(* Chamber *)
IF Config.ChamberConfigs.PhotoLumChamberConfig.IsEnabled THEN
	Chamber.FB_init(FALSE, FALSE, Config := Config.ChamberConfigs.PhotoLumChamberConfig);	
END_IF

// Chuck
IF Config.ChuckConfigs.PhotoLumChuckConfig.IsEnabled THEN
	Chuck.FB_init(FALSE, FALSE, Config := Config.ChuckConfigs.PhotoLumChuckConfig);	
END_IF 

// Axis
IF Config.AxesConfigs.Ps10OwisAxisConfig.IsEnabled THEN
	Ps10Axis.FB_init(FALSE, FALSE, Config := Config.AxesConfigs.Ps10OwisAxisConfig);	
END_IF

(* LightConfigs *) 
IF Config.LightConfigs.EvosensLightConfig.IsEnabled THEN
	EvosensLight.FB_init(FALSE, FALSE, Config := Config.LightConfigs.EvosensLightConfig);
ELSIF Config.LightConfigs.ArduinoLightConfig.IsEnabled THEN
	ArduinoLight.FB_init(FALSE, FALSE, Config := Config.LightConfigs.ArduinoLightConfig);	
END_IF

(* DistanceSensorConfigs *) 
IF Config.DistanceSensorConfigs.MicroEpsilonDistanceSensorConfig.IsEnabled THEN
	MicroEpsilonDistanceSensor.FB_init(FALSE, FALSE, Config := Config.DistanceSensorConfigs.MicroEpsilonDistanceSensorConfig);	
END_IF

IF Config.IsEnabled THEN
	_logger.Information('PhotoLum devices initialization ended...');
END_IF
END_METHOD

END_FUNCTION_BLOCK

// ---- PMShared/Hardware/Devices/Chambers/PhotoLum/PhotoLumChamber.TcPOU
{attribute 'OPC.UA.DA' := '1'}
FUNCTION_BLOCK PhotoLumChamber EXTENDS ChamberBase
VAR_INPUT
	IoChamberPhotoLum : IoChamberPhotoLum;
END_VAR
VAR_OUTPUT
END_VAR
VAR
	{attribute 'OPC.UA.DA' := '0'}
	_config : PhotoLumChamberConfig;	
	
	{attribute 'OPC.UA.DA' := '0'}
	_initDevice : BOOL;
	
	{attribute 'OPC.UA.DA' := '0'}
	_itemInit : INT;
	{attribute 'OPC.UA.DA' := '0'}
	_itemScheduler : INT;
	{attribute 'OPC.UA.DA' := '0'}
	_itemExecScheduler : INT;		
	{attribute 'OPC.UA.DA' := '0'}
	_itemRaisedProperties : INT;			
	{attribute 'OPC.UA.DA' := '0'}
	_pulseGenerator : TON;	
	
	{region 'Commands'}	
		 	
	{attribute 'OPC.UA.DA' := '0'}
	_enableCamera : BOOL;
	{attribute 'OPC.UA.DA' := '0'}
	_moveSlitDoorPositionCmd	 : BOOL;	
	{attribute 'OPC.UA.DA' := '0'}			  		   
	_raisePropertiesCmd : BOOL;	 
			
	{endregion}
	
	{attribute 'OPC.UA.DA' := '0'}
	_deliverMessages : INT;
	
	InterlockPanelsMsg : STRING(255);
	SlitDoorPositionMsg : STRING(255);
	SlitDoorOpenPositionMsg : STRING(255);
	SlitDoorClosePositionMsg : STRING(255);
	
	{attribute 'OPC.UA.DA' := '0'}
	message : STRING(255);
	
	{attribute 'OPC.UA.DA' := '0'}
	_pos : INT;	
	
	{attribute 'OPC.UA.DA' := '0'}
	tmpConcat1 : STRING;
	{attribute 'OPC.UA.DA' := '0'}
	tmpConcat2 : STRING;
	{attribute 'OPC.UA.DA' := '0'}
	tmpConcatName : STRING; 
	{attribute 'OPC.UA.DA' := '0'}
	tmpConcatDescription : STRING;
	{attribute 'OPC.UA.DA' := '0'}
	tmpConcatInterlockID : STRING;
	
	{attribute 'OPC.UA.DA' := '0'}
	_itemInterlock : UINT;
	{attribute 'OPC.UA.DA' := '0'}
	_interlockCount : UINT;			
END_VAR

SUPER^();

// Init device
InitDevice(); 

// Deliver messages
CASE _deliverMessages OF	
	EFeedbackMsgPhotoLumChamber.InterlockPanelsMsg :
		InterlockPanelsMsg := message;	
	EFeedbackMsgPhotoLumChamber.SlitDoorPositionMsg :
		SlitDoorPositionMsg := TO_STRING(SlitDoorPosition);		
	EFeedbackMsgPhotoLumChamber.SlitDoorOpenPositionMsg :
		SlitDoorOpenPositionMsg := TO_STRING(SlitDoorOpenPosition);	
	EFeedbackMsgPhotoLumChamber.SlitDoorClosePositionMsg :
		SlitDoorClosePositionMsg := TO_STRING(SlitDoorClosePosition);		
END_CASE

// Commands
MoveSlitDoorPosition(_moveSlitDoorPositionCmd, _pos); 
RaisePropertiesChanged(_raisePropertiesCmd);

IF NOT _moveSlitDoorPositionCmd AND NOT _raisePropertiesCmd THEN	
	MessageScheduler();
END_IF

METHOD FB_init : BOOL
VAR_INPUT
	bInitRetains : BOOL; // if TRUE, the retain variables are initialized (warm start / cold start)
	bInCopyCode : BOOL;  // if TRUE, the instance afterwards gets moved into the copy code (online change)
	Config : PhotoLumChamberConfig;
END_VAR
IF Config.IsEnabled THEN
	_config := Config;	

	SUPER^._chamberConfig.Name := Config.Name;
	SUPER^._chamberConfig.DeviceID := Config.DeviceID;
	SUPER^._chamberConfig.IsEnabled := Config.IsEnabled;
	SUPER^._chamberConfig.LogLevel := Config.LogLevel;
	
	SUPER^.Name := Config.Name;
	SUPER^.DeviceID := Config.DeviceID;
	
	THIS^.Family := DeviceFamily.Chamber;

	THIS^.SetReady();
	_Logger.Information(_message.Reset().Append('Init ').
							Append('{').Append(TO_STRING(THIS^.Family)).Append('} - ').
							Append('{').Append(TO_STRING(THIS^.Name)).Append('} - ').
							Append('Status : ').Append(TO_STRING(THIS^.Status)).
							ToString());										 
END_IF
END_METHOD

METHOD InitDevice
VAR_INPUT
END_VAR
IF NOT _initDevice THEN			
	_logger.Information(_message.Reset().
								Append(_config.Name).
								Append(' - init device').ToString());		
							
	_initDevice := TRUE;
	
END_IF
END_METHOD

METHOD MessageScheduler
VAR_INPUT
END_VAR
IF _pulseGenerator.Q THEN
	_pulseGenerator(IN := FALSE, PT := T#10MS);
		
	CASE _itemScheduler OF	
		0: SlitDoorPositionMsg := ' ';
		   _itemScheduler := 1;
		   
		1: ReadInterlock();
		   _itemScheduler := 2;
	
		2:  ReadSlitDoorPosition();
			_itemScheduler := 3;

		3:  ReadSlitDoorOpenPosition();
			_itemScheduler := 4;

		4:  ReadSlitDoorClosePosition();
			_itemScheduler := 0;					
	END_CASE
ELSE
	_pulseGenerator(IN := TRUE, PT := T#50MS);		
END_IF
END_METHOD

{attribute 'TcRpcEnable' := '1'}
METHOD MoveSlitDoorPosition
VAR_INPUT
	Execute : BOOL;
	Position : INT;
END_VAR
IF Execute THEN
	_logger.Information(_message.Reset().Append(_config.Name).Append(' - Move slit door position : ').Append(TO_STRING(Position)).ToString());
	
	_moveSlitDoorPositionCmd := FALSE;
		
	IF Position = ESlitDoorPosition.Open THEN
		IoChamberPhotoLum.OutputOpenSlitDoor := TRUE;
		IoChamberPhotoLum.OutputCloseSlitDoor := FALSE;
	ELSIF Position = ESlitDoorPosition.Close THEN
		IoChamberPhotoLum.OutputOpenSlitDoor := FALSE;
		IoChamberPhotoLum.OutputCloseSlitDoor := TRUE;
		
		//IsInLoadingPosition := FALSE;
	ELSE
		_logger.Error(_message.Reset().Append(_config.Name).Append(' - unknown position : ').Append(TO_STRING(Position)).ToString());
		
		//IsInLoadingPosition := FALSE;
	END_IF
				
	_itemScheduler := 0;
END_IF
END_METHOD

{attribute 'TcRpcEnable' := '1'}
METHOD RaisePropertiesChanged
VAR_INPUT
	Execute : BOOL;
END_VAR
IF Execute THEN		
	_raisePropertiesCmd := TRUE;	
		
	IF _pulseGenerator.Q THEN
		_pulseGenerator(IN := FALSE, PT := T#10MS);
		
		CASE _itemRaisedProperties OF		
			0: 	SUPER^._raisePropertiesBase := TRUE;		   
				_itemRaisedProperties := 10;
				
			10: _logger.Information(_message.Reset().Append(_config.Name).Append(' - RaisePropertiesChanged').ToString());
				_raisePropertiesCmd := FALSE;
				_itemRaisedProperties := 0;
		END_CASE	
	ELSE
		_pulseGenerator(IN := TRUE, PT := T#50MS);	
	END_IF		
END_IF
END_METHOD

METHOD ReadInterlock 
VAR_INPUT
END_VAR
VAR
	statePanel : STRING;
END_VAR
_deliverMessages := EFeedbackMsgPsdChamber.InterlockPanelsMsg;

IF _interlockCount < Const.PHOTOLUM_NUMBER_INTERLOCK_PANELS - 1 THEN
	_interlockCount := _interlockCount + 1;
ELSE
	_interlockCount := 0;
END_IF

tmpConcatName := CONCAT(_config.Interlock[_interlockCount].Name, ';');
tmpConcatDescription := CONCAT(_config.Interlock[_interlockCount].Description, ';');
tmpConcatInterlockID := CONCAT(UINT_TO_STRING(_config.Interlock[_interlockCount].InterlockID), ';');

tmpConcat1 := CONCAT(tmpConcatName, tmpConcatDescription);
tmpConcat2 := CONCAT(tmpConcat1, tmpConcatInterlockID);

IF _config.Interlock[_interlockCount].State THEN
	statePanel := 'Closed';
ELSE
	statePanel := 'Opened';
END_IF

message := CONCAT(tmpConcat2, statePanel);
END_METHOD

METHOD ReadSlitDoorClosePosition
VAR_INPUT
END_VAR
VAR
	open : BOOL;
	close : BOOL;
END_VAR
_deliverMessages := EFeedbackMsgPhotoLumChamber.SlitDoorClosePositionMsg;
SlitDoorClosePosition := IoChamberPhotoLum.InputCloseSlitDoor;
END_METHOD

METHOD ReadSlitDoorOpenPosition
VAR_INPUT
END_VAR
_deliverMessages := EFeedbackMsgPhotoLumChamber.SlitDoorOpenPositionMsg;
SlitDoorOpenPosition := IoChamberPhotoLum.InputOpenSlitDoor;
END_METHOD

METHOD ReadSlitDoorPosition
VAR_INPUT
END_VAR
VAR
	open : BOOL;
	close : BOOL;
END_VAR
_deliverMessages := EFeedbackMsgPhotoLumChamber.SlitDoorPositionMsg;

open := IoChamberPhotoLum.InputOpenSlitDoor;
close := IoChamberPhotoLum.InputCloseSlitDoor;

IF open AND NOT close THEN
	IoChamberPhotoLum.EfemInterlockSlitDoor := TRUE;	
	IoChamberPhotoLum.EfemInterlockArmExtendedEnable := TRUE;	
	SlitDoorPosition := ESlitDoorPosition.Open;	
ELSIF close AND NOT open THEN
	IoChamberPhotoLum.EfemInterlockSlitDoor := FALSE;
	IoChamberPhotoLum.EfemInterlockArmExtendedEnable := FALSE;
	SlitDoorPosition := ESlitDoorPosition.Close;
ELSIF close AND open THEN
	IoChamberPhotoLum.EfemInterlockSlitDoor := FALSE;
	IoChamberPhotoLum.EfemInterlockArmExtendedEnable := FALSE;
	SlitDoorPosition := ESlitDoorPosition.Error;	
ELSE
	IoChamberPhotoLum.EfemInterlockSlitDoor := FALSE;
	IoChamberPhotoLum.EfemInterlockArmExtendedEnable := FALSE;
	SlitDoorPosition := ESlitDoorPosition.Unknown;		
END_IF
END_METHOD

END_FUNCTION_BLOCK

// ---- PMShared/Hardware/Devices/Chucks/PhotoLum/PhotoLumChuck.TcPOU
FUNCTION_BLOCK PhotoLumChuck EXTENDS ChuckBase
VAR_INPUT
	IoChuck : IoChuckPhotoLum;
END_VAR
VAR_OUTPUT
END_VAR
VAR
	{attribute 'OPC.UA.DA' := '0'}
	_config : PhotoLumChuckConfig;
	
	{attribute 'OPC.UA.DA' := '0'}
	_deliverMessages : INT;
	
	WaferPresenceMsg : STRING(255);
	
	{attribute 'OPC.UA.DA' := '0'}
	_initDevice : BOOL;
	
	{attribute 'OPC.UA.DA' := '0'}
	_itemInit : INT;
	
	{attribute 'OPC.UA.DA' := '0'}
	_itemScheduler : INT;
	{attribute 'OPC.UA.DA' := '0'}
	_itemRaisedProperties : INT;
	{attribute 'OPC.UA.DA' := '0'}
	_pulseGenerator : TON;
	
	{region 'Commands'}
		
	{attribute 'OPC.UA.DA' := '0'}			  		   
	_clampWaferCmd : BOOL;
	{attribute 'OPC.UA.DA' := '0'}			  		   
	_releaseWaferCmd : BOOL;
	{attribute 'OPC.UA.DA' := '0'}			  		   
	_raisePropertiesCmd : BOOL;
			
	{endregion}	
		
	{attribute 'OPC.UA.DA' := '0'}	
	_size : LREAL;	
		 
	{attribute 'OPC.UA.DA' := '0'}
	message : STRING;
	{attribute 'OPC.UA.DA' := '0'}
	_waferPresenceSensorCounter : UINT;			
	
	
	
END_VAR

SUPER^();

// Init device
InitDevice(); 

// Deliver messages
CASE _deliverMessages OF		
	EFeedbackMsgPhotoLumChuck.WaferPresenceMsg :
		WaferPresenceMsg := message;		
END_CASE
	
_deliverMessages := 0;

// Commands	
ClampWafer(_clampWaferCmd, _size);
ReleaseWafer(_releaseWaferCmd, _size);
RaisePropertiesChanged(_raisePropertiesCmd);

IF (NOT _raisePropertiesCmd) THEN
	MessageScheduler();
END_IF

{attribute 'TcRpcEnable' := '1'}
METHOD ClampWafer
VAR_INPUT
	Execute : BOOL;
	Value : LREAL;
END_VAR
VAR 
	size : EWaferSize := EWaferSize.Unknown;
END_VAR
IF Execute THEN
	_logger.Information(_message.Reset().Append(_config.Name).Append(' - Clamp wafer: ').Append(TO_STRING(Value)).ToString());

	CASE LREAL_TO_INT(Value) OF
		EWaferSize._100mm : 
			IoChuck.OutputVaccum100mm := TRUE;
			IoChuck.OutputVaccum150mm := FALSE; 
			IoChuck.OutputVaccum200mm := FALSE;			
			size := EWaferSize._100mm;
			
		EWaferSize._150mm :
			IoChuck.OutputVaccum100mm := FALSE;
			IoChuck.OutputVaccum150mm := TRUE; 
			IoChuck.OutputVaccum200mm := FALSE;
			size := EWaferSize._150mm;
			
		EWaferSize._200mm :
			IoChuck.OutputVaccum100mm := FALSE;
			IoChuck.OutputVaccum150mm := FALSE; 
			IoChuck.OutputVaccum200mm := TRUE;
			size := EWaferSize._200mm;
			
		EWaferSize.Unknown:		
			size := EWaferSize.Unknown;
			_logger.Warning(_message.Reset().Append(_config.Name).Append(' - Unknown size ').ToString());
	ELSE 
		_logger.Warning(_message.Reset().Append(_config.Name).Append(' - This size: ').Append(TO_STRING(Value)).Append(' does not exist').ToString());
	END_CASE
	
	WaferSize := size;
	
	_clampWaferCmd := FALSE;
END_IF
END_METHOD

METHOD FB_init : BOOL
VAR_INPUT
	bInitRetains : BOOL; // if TRUE, the retain variables are initialized (warm start / cold start)
	bInCopyCode : BOOL;  // if TRUE, the instance afterwards gets moved into the copy code (online change)
	Config : PhotoLumChuckConfig;
END_VAR
IF Config.IsEnabled THEN
	_config := Config;
	
	SUPER^._chuckConfig.Name := Config.Name;
	SUPER^._chuckConfig.DeviceID := Config.DeviceID;
	SUPER^._chuckConfig.IsEnabled := Config.IsEnabled;
	SUPER^._chuckConfig.LogLevel := Config.LogLevel;
	
	SUPER^.Name := Config.Name;
	SUPER^.DeviceID := Config.DeviceID;
	
	THIS^.Family := DeviceFamily.Chuck;

	THIS^.SetReady();
	_Logger.Information(_message.Reset().Append('Init ').
							Append('{').Append(TO_STRING(THIS^.Family)).Append('} - ').
							Append('{').Append(TO_STRING(THIS^.Name)).Append('} - ').
							Append('Status : ').Append(TO_STRING(THIS^.Status)).
							ToString());										 
END_IF
END_METHOD

METHOD InitDevice
VAR_INPUT
END_VAR
IF NOT _initDevice THEN			
	_logger.Information(_message.Reset().
								Append(_config.Name).
								Append(' - init device').ToString());		
								
	_initDevice := TRUE;
END_IF
END_METHOD

METHOD MessageScheduler
VAR_INPUT
END_VAR
IF _pulseGenerator.Q THEN
	_pulseGenerator(IN := FALSE, PT := T#10MS);
		
	CASE _itemScheduler OF	
		0:	WaferPresenceMsg := ' ';
			_itemScheduler := 1;
	
		1:	ReadWaferPresence();
			_itemScheduler := 0;		
									
	END_CASE
ELSE
	_pulseGenerator(IN := TRUE, PT := T#100MS);	
END_IF
END_METHOD

{attribute 'TcRpcEnable' := '1'}
METHOD RaisePropertiesChanged
VAR_INPUT
	Execute : BOOL;
END_VAR
IF Execute THEN		
	_raisePropertiesCmd := TRUE;	
	
	IF _pulseGenerator.Q THEN
		_pulseGenerator(IN := FALSE, PT := T#10MS);
		
		CASE _itemRaisedProperties OF		
			0: _itemRaisedProperties := 10;
				
			10: _logger.Information(_message.Reset().Append(_config.Name).Append(' - RaisePropertiesChanged').ToString());
				_raisePropertiesCmd := FALSE;
				_itemRaisedProperties := 0;		
		END_CASE	
	ELSE
		_pulseGenerator(IN := TRUE, PT := T#100MS);	
	END_IF		
END_IF
END_METHOD

METHOD ReadWaferPresence
VAR_INPUT
END_VAR
VAR	
	waferPresence : STRING;
	diameter : STRING;
END_VAR
_deliverMessages := EFeedbackMsgPsdChuck.WaferPresenceMsg;

IF _waferPresenceSensorCounter < Const.PHOTOLUM_NUMBER_WAFER_PRESENCE_SENSORS - 1 THEN
	_waferPresenceSensorCounter := _waferPresenceSensorCounter + 1;
ELSE
	_waferPresenceSensorCounter := 0;
END_IF

diameter := TO_STRING(_config.WaferPresenceSensor[_waferPresenceSensorCounter].Diameter);

IF _config.WaferPresenceSensor[_waferPresenceSensorCounter].InputWaferPresence AND 
   _config.WaferPresenceSensor[_waferPresenceSensorCounter].Diameter = TO_UINT(_waferSize) THEN
	waferPresence := INT_TO_STRING(EMaterialPresence.Present);
ELSE
	waferPresence := INT_TO_STRING(EMaterialPresence.NotPresent);		
END_IF

message := CONCAT(CONCAT(diameter, ';'), waferPresence);
END_METHOD

{attribute 'TcRpcEnable' := '1'}
METHOD ReleaseWafer
VAR_INPUT
	Execute : BOOL;
	Value : LREAL;
END_VAR
IF Execute THEN
	_logger.Information(_message.Reset().Append(_config.Name).Append(' - release wafer: ').Append(TO_STRING(Value)).ToString());

	IF Value = EWaferSize._100mm THEN
		IoChuck.OutputVaccum100mm := FALSE;
	ELSIF Value = EWaferSize._150mm THEN		
		IoChuck.OutputVaccum150mm := FALSE; 		
	ELSIF Value = EWaferSize._200mm THEN
		IoChuck.OutputVaccum200mm := FALSE;
	ELSIF Value = EWaferSize.Unknown THEN
		_logger.Warning(_message.Reset().Append(_config.Name).Append(' - Unknown size ').ToString());
	ELSE 
		_logger.Warning(_message.Reset().Append(_config.Name).Append(' - This size: ').Append(TO_STRING(Value)).Append(' does not exist').ToString());
	END_IF

	WaferSize := EWaferSize.Unknown;
	
	_releaseWaferCmd := FALSE;
END_IF
END_METHOD

END_FUNCTION_BLOCK

// ---- PMShared/Hardware/Devices/Axes/Owis/Ps10Axis.TcPOU
FUNCTION_BLOCK Ps10Axis EXTENDS AxesBase
VAR_INPUT
END_VAR
VAR_OUTPUT
END_VAR
VAR
	{attribute 'OPC.UA.DA' := '0'}
	_config : Ps10OwisAxisConfig;
	{attribute 'OPC.UA.DA' := '0'}
	_coeAccess : CoeAccess;
	{attribute 'OPC.UA.DA' := '0'}
	_initConfigSerialCom : BOOL;	
	{attribute 'OPC.UA.DA' := '0'}
	_serialCom  : SerialCom(Prefix :='', Suffix := Const.CARRIAGE_RETURN);
	{attribute 'OPC.UA.DA' := '0'}
	_refSerialCom : REFERENCE TO SerialCom(Prefix :='', Suffix := Const.CARRIAGE_RETURN) := _serialCom;	 
	{attribute 'OPC.UA.DA' := '0'}
	_isReceived : BOOL;
	
	{attribute 'OPC.UA.DA' := '0'}
	_deliverMessages : INT;
	
	StatusMsg : STRING(255);
	AxisStatusMsg : STRING(255);
	DrivingCurrentMsg : STRING(255);
	HoldingCurrentMsg : STRING(255);
	LimitSwitchtMsg : STRING(255);
	ErrMsg : STRING(255);
	PositionMsg : STRING(255);
	CustomMsg : STRING(255);
	IsInMovingMsg : STRING(255);
	
	{region 'Commands'}	

	{attribute 'OPC.UA.DA' := '0'}
	_cmdConfigDeviceParameters : BOOL;
	{attribute 'OPC.UA.DA' := '0'}
	_cmdClearErr : BOOL;
	{attribute 'OPC.UA.DA' := '0'}
	_cmdMotorInit : BOOL;
	{attribute 'OPC.UA.DA' := '0'}
	_cmdDrivingCurrent : BOOL;
	{attribute 'OPC.UA.DA' := '0'}
	_cmdHoldingCurrent : BOOL;
	{attribute 'OPC.UA.DA' := '0'}	 
	_cmdLimitSwitch : BOOL;
	{attribute 'OPC.UA.DA' := '0'}
	_cmdReset : BOOL;
	{attribute 'OPC.UA.DA' := '0'}
	_cmdStopMotion : BOOL;		 
	{attribute 'OPC.UA.DA' := '0'}
	_cmdHomePosition : BOOL;
	{attribute 'OPC.UA.DA' := '0'}
	_cmdMoveAbsPosition : BOOL;
	{attribute 'OPC.UA.DA' := '0'}
	_customCmd : BOOL;
	{attribute 'OPC.UA.DA' := '0'}			  		   
	_cmdRaiseProperties : BOOL;	 
			
	{endregion}
		 
	{attribute 'OPC.UA.DA' := '0'}
	_initDevice : BOOL;	
		
	{attribute 'OPC.UA.DA' := '0'}
	_posToDegree : LREAL;
	{attribute 'OPC.UA.DA' := '0'}
	_cmd : STRING;
	{attribute 'OPC.UA.DA' := '0'}
	_itemScheduler : INT;
	{attribute 'OPC.UA.DA' := '0'}
	_itemRaisedProperties : INT;
	{attribute 'OPC.UA.DA' := '0'}
	_itemMove : INT;	
	{attribute 'OPC.UA.DA' := '0'}
	_itemInit : INT;
	{attribute 'OPC.UA.DA' := '0'}
	_itemdConfigDeviceParameters : INT;
	{attribute 'OPC.UA.DA' := '0'}
	_pulseGenerator : TON;
	{attribute 'OPC.UA.DA' := '0'}
	_pulseMoveGenerator : TON;	
	{attribute 'OPC.UA.DA' := '0'}
	_initPulseGenerator : TON;	
	{attribute 'OPC.UA.DA' := '0'}	
	_execPulseGenerator : TON;
	{attribute 'OPC.UA.DA' := '0'}	
	_configDeviceParamsPulseGenerator : TON;	
	
	{attribute 'OPC.UA.DA' := '0'}
	message : STRING;
	{attribute 'OPC.UA.DA' := '0'}
	lastMessage : STRING;	
	{attribute 'OPC.UA.DA' := '0'}
	stringLength : INT;
	{attribute 'OPC.UA.DA' := '0'}
	_convertDegreeToCount : LREAL := 83;
	{attribute 'OPC.UA.DA' := '0'}
	_currentAxisMode : STRING;
	{attribute 'OPC.UA.DA' := '0'}
	_currentPos : LREAL;	
	{attribute 'OPC.UA.DA' := '0'} 
	_currentPositionCounter : UINT;
	{attribute 'OPC.UA.DA' := '0'} 
	_isInMoving : BOOL;
END_VAR

IF NOT InitConfigSerialCom THEN
	ConfigureSerialCom();
ELSIF THIS^.Status = TExecutionState.Ready THEN				
	IF _refSerialCom.ErrorReceiveId = COMERROR_NOERROR THEN
		_refSerialCom(TxBuffer:= HardwareGlobalVariables.TxBufferFilterWheel, 
		 	      	  RxBuffer:= HardwareGlobalVariables.RxBufferFilterWheel);
	END_IF			

	// Init device	
	InitDevice();
		 				  	
	// Deliver messages
	IF _refSerialCom.IsReceived THEN		
		lastMessage := _refSerialCom.LastReceivedString;			
		stringLength := LEN(lastMessage);
		
		IF stringLength > 1 THEN
			message := LEFT(lastMessage, stringLength - 1);
		ELSE
			message := ' ';
		END_IF; 
				
		CASE _deliverMessages OF	
			EFeedbackMsgOwisPs10.AxisStateMsg :
				_currentAxisMode := MID(message, 1, STRING_TO_INT(AxesConst.AXIS_FILTER_WHEEL));
				AxisStatusMsg := ParseAxisStatus(_currentAxisMode);
			EFeedbackMsgOwisPs10.DrivingCurrentMsg :
				 DrivingCurrentMsg := message;
			EFeedbackMsgOwisPs10.HoldingCurrentMsg :
				 HoldingCurrentMsg := message;
			EFeedbackMsgOwisPs10.LimitSwitchMsg :
				 LimitSwitchtMsg := message;
			EFeedbackMsgOwisPs10.ErrMsg :
				 ErrMsg := message;
			EFeedbackMsgOwisPs10.PositionMsg :					
				_currentPos := STRING_TO_LREAL(message) / _convertDegreeToCount;
				PositionMsg := LREAL_TO_STRING(_currentPos);				
			EFeedbackMsgOwisPs10.CurrentPositionCounterMsg :
				_currentPositionCounter := STRING_TO_UINT(message);			
			EFeedbackMsgOwisPs10.CustomMsg :
				CustomMsg := message;						
			END_CASE
	END_IF		
			
	IF (_initDevice AND NOT _cmdClearErr AND NOT _cmdMotorInit AND NOT _cmdConfigDeviceParameters AND NOT _cmdDrivingCurrent AND NOT 
		_cmdHoldingCurrent AND NOT _cmdLimitSwitch AND NOT _cmdStopMotion AND NOT _cmdHomePosition AND NOT _cmdMoveAbsPosition AND NOT 
		_customCmd AND NOT _cmdRaiseProperties) THEN
			MessageScheduler();
	END_IF
	
	ConfigDeviceParameters(_cmdConfigDeviceParameters);
	ClearError(_cmdClearErr);
	MotorInit(_cmdMotorInit);
	SetDrivingCurrent(_cmdDrivingCurrent);
	SetHoldingCurrent(_cmdHoldingCurrent);
	SetLimitSwitch(_cmdLimitSwitch);
	Reset(_cmdReset);
	StopMotion(_cmdStopMotion);
	HomePosition(_cmdHomePosition);	
	MoveAbsPosition(_cmdMoveAbsPosition, _posToDegree);
	CustomCommand(_customCmd, _cmd);	
	RaisePropertiesChanged(_cmdRaiseProperties);	
	
END_IF

{attribute 'TcRpcEnable' := '1'}
METHOD ClearError
VAR_INPUT
	Execute : BOOL;
END_VAR
VAR
	cmd : STRING := 'ERRCLEAR';
END_VAR
IF Execute THEN
	_logger.Information(_message.Reset().Append(_config.Name).Append(' - Clear error').ToString());
	_serialCom.Send(cmd);	

	_cmdClearErr := FALSE;
END_IF
END_METHOD

METHOD ConfigDeviceParameters
VAR_INPUT
	Execute : BOOL;
END_VAR
VAR	
END_VAR
IF Execute THEN

	_cmdConfigDeviceParameters := TRUE;	

	IF _configDeviceParamsPulseGenerator.Q THEN
		_configDeviceParamsPulseGenerator(IN := FALSE, PT := T#10MS);
		
		CASE _itemdConfigDeviceParameters OF
			0:  _logger.Information(_message.Reset().Append(_config.Name).Append(' - Configure device parameters').ToString());
				_itemdConfigDeviceParameters := 1;				
								
			1: _cmdDrivingCurrent := TRUE;
				_itemdConfigDeviceParameters := 2;

			2: _cmdHoldingCurrent := TRUE;
				_itemdConfigDeviceParameters := 3;				
			
			3: _cmdLimitSwitch := TRUE;
				_itemdConfigDeviceParameters := 4;	
			
			4: _cmdMotorInit := TRUE;
				_itemdConfigDeviceParameters := 5;					
				
			5: _logger.Information(_message.Reset(). Append(_config.Name). Append(' - Configure device parameters done').ToString());	
			   _itemdConfigDeviceParameters := 0;			
			   _cmdConfigDeviceParameters := FALSE;
		END_CASE
	ELSE
		_configDeviceParamsPulseGenerator(IN := TRUE, PT := T#200MS);		
	END_IF		
END_IF
END_METHOD

METHOD ConfigureSerialCom
VAR_INPUT
END_VAR
IF _coeAccess.CoeOperation.Ready THEN
	_logger.Information(_message.Reset().Append('Start configuration com serial').ToString());
END_IF;	

_coeAccess.CoeOperation.Start();
_coeAccess(SerialCommunication := _config.SerialCommunication);
	
IF _coeAccess.CoeOperation.Done THEN
	_coeAccess.SetDone();	
 
	_Logger.Information(_message.Reset().
							Append('{').Append(TO_STRING(THIS^.Family)).Append('} : ').
							Append(' - Status : ').Append(TO_STRING(_coeAccess.Status)).ToString());	
	InitConfigSerialCom := TRUE;
END_IF
 
IF _coeAccess.CoeOperation.Error THEN	
	_coeAccess.SetError(0);
	
	_Logger.Error(_message.Reset().
							Append('{').Append(TO_STRING(THIS^.Family)).Append('} : ').
							Append(' - Status : ').Append(TO_STRING(_coeAccess.Status)).ToString());
	InitConfigSerialCom := TRUE;
END_IF

THIS^.Status := _coeAccess.Status;
State := _coeAccess.Status;
END_METHOD

{attribute 'TcRpcEnable' := '1'}
METHOD CustomCommand
VAR_INPUT
	Execute : BOOL;
	Cmd : STRING;
END_VAR
IF Execute THEN
	_logger.Information(_message.Reset().Append(_config.Name).Append(' - Custom : ').Append(Cmd).ToString());
	_deliverMessages := EFeedbackMsgOwisPs10.CustomMsg;									
	_serialCom.Send(Cmd);
	
	_customCmd := FALSE;
END_IF
END_METHOD

{attribute 'TcRpcEnable' := '1'}
METHOD ErrorMessages
VAR_INPUT
END_VAR
VAR
	cmd : STRING := '?MSG';
END_VAR
_deliverMessages := EFeedbackMsgOwisPs10.ErrMsg;	
_serialCom.Send(cmd);
END_METHOD

METHOD FB_init : BOOL
VAR_INPUT
	bInitRetains : BOOL; // if TRUE, the retain variables are initialized (warm start / cold start)
	bInCopyCode : BOOL;  // if TRUE, the instance afterwards gets moved into the copy code (online change)
	Config : Ps10OwisAxisConfig;
END_VAR
IF Config.IsEnabled THEN
	_config := Config;
	
	SUPER^._axisConfig.Name := Config.Name;
	SUPER^._axisConfig.DeviceID := Config.DeviceID;
	SUPER^._axisConfig.IsEnabled := Config.IsEnabled;
	SUPER^._axisConfig.LogLevel := Config.LogLevel;
	
	SUPER^.Name := Config.Name;
	SUPER^.DeviceID := Config.DeviceID;	
	THIS^.Family := DeviceFamily.Axes;
	
	_Logger.Information(_message.Reset().Append('Init ').
							Append('{').Append(TO_STRING(THIS^.Family)).Append('} - ').
							Append('{').Append(TO_STRING(Config.Name)).Append('}').ToString());																													
END_IF
END_METHOD

(** Axis state inquiry **)
METHOD GetAxisStatus : STRING
VAR_INPUT
END_VAR
VAR
	cmd : STRING := '?ASTAT';
END_VAR
_deliverMessages := EFeedbackMsgOwisPs10.AxisStateMsg;	
_serialCom.Send(cmd);
END_METHOD

(** Read out driving current with stepper motors in percent **)
METHOD PROTECTED GetDrivingCurrent
VAR_INPUT
END_VAR
VAR
	cmd : STRING := '?DRICUR';
END_VAR
_deliverMessages := EFeedbackMsgOwisPs10.DrivingCurrentMsg;	
_serialCom.Send(Concat(cmd, AxesConst.AXIS_FILTER_WHEEL));
END_METHOD

(** Read out holding current with stepper motor axis in percent **)
METHOD PROTECTED GetHoldingCurrent
VAR_INPUT
END_VAR
VAR
	cmd : STRING := '?HOLCUR';
END_VAR
_deliverMessages := EFeedbackMsgOwisPs10.HoldingCurrentMsg;	
_serialCom.Send(Concat(cmd, AxesConst.AXIS_FILTER_WHEEL));
END_METHOD

(** Read out limit switch mask for the axis **)
METHOD PROTECTED GetLimitSwitch
VAR_INPUT
END_VAR
VAR
	cmd : STRING := '?SMK';
END_VAR
_deliverMessages := EFeedbackMsgOwisPs10.LimitSwitchMsg;	
_serialCom.Send(Concat(cmd, AxesConst.AXIS_FILTER_WHEEL));
END_METHOD

(** Position Query **)
METHOD PROTECTED GetPosition
VAR_INPUT
END_VAR
VAR
	cmd : STRING := '?PSET';
END_VAR
_deliverMessages := EFeedbackMsgOwisPs10.PositionMsg;	
_serialCom.Send(Concat(cmd, AxesConst.AXIS_FILTER_WHEEL));
END_METHOD

{attribute 'TcRpcEnable' := '1'}
METHOD HomePosition
VAR_INPUT
	Execute : BOOL;
END_VAR
VAR
	cmd : STRING := 'REF';
END_VAR
IF Execute THEN	
	_logger.Information(_message.Reset().Append(_config.Name).Append(' - Home position : ').ToString());
	cmd := Concat(CONCAT(cmd, AxesConst.AXIS_FILTER_WHEEL), '=');	
	_serialCom.Send(Concat(cmd, '4'));
	
	_cmdHomePosition := FALSE;
END_IF
END_METHOD

PROPERTY InitConfigSerialCom : BOOL
GET
InitConfigSerialCom := _initConfigSerialCom;
END_GET
SET
_initConfigSerialCom := InitConfigSerialCom;
END_SET
END_PROPERTY

METHOD InitDevice
VAR_INPUT
END_VAR
VAR
	displayingPositionCmd : STRING := 'PWMSMODE';
	absoluteModeCmd : STRING := 'ABSOL';
	
	displayingPositionInDegree : STRING;
END_VAR
IF NOT _initDevice THEN	
	IF _initPulseGenerator.Q THEN
		_initPulseGenerator(IN := FALSE, PT := T#10MS);
		
		CASE _itemInit OF
			0:  _logger.Information(_message.Reset().Append(_config.Name).Append(' - InitDevice').ToString());
				_itemInit := 1;				
				
			1:  _cmdClearErr := TRUE;
				_itemInit := 2;
			
			2: // Absolute mode
				_serialCom.Send(CONCAT(absoluteModeCmd, AxesConst.AXIS_FILTER_WHEEL));	
				_itemInit := 10;
				
			10: _cmdConfigDeviceParameters := TRUE;	
			   _itemInit := 11;
			
			11: IF NOT _cmdConfigDeviceParameters THEN
					_itemInit := 20;
				END_IF
			
			20: GetAxisStatus();
				_itemInit := 21;
				
			21: // Displaying position in °
				displayingPositionInDegree := Concat(CONCAT(displayingPositionCmd, AxesConst.AXIS_FILTER_WHEEL), '=');
				_serialCom.Send(CONCAT(displayingPositionInDegree, '3'));				
				_itemInit := 22;													
				
			22:  IF _currentAxisMode = 'R' THEN	
					_itemInit := 30;	
				ELSE			
					_logger.Error(_message.Reset().Append(_config.Name).Append(' - Axis status : ').
								  Append(_currentAxisMode).ToString());
					_itemInit := 40;				  
			    END_IF							
				
			30:  GetPosition();
				_itemInit := 31;	
				
			31: _posToDegree := _currentPos;
				_itemInit := 40;
				
			40: _logger.Information(_message.Reset(). Append(_config.Name). Append(' - InitDevice done').ToString());	
				_itemInit := 0;			
				_initDevice	:= TRUE;
		END_CASE
	ELSE
		_initPulseGenerator(IN := TRUE, PT := T#100MS);		
	END_IF		
END_IF
END_METHOD

PROPERTY IsInMoving : bool
GET
IsInMoving := _isInMoving;
END_GET
SET
_isInMoving := IsInMoving;
END_SET
END_PROPERTY

METHOD MessageScheduler
VAR_INPUT
END_VAR
IF _pulseGenerator.Q THEN
	_pulseGenerator(IN := FALSE, PT := T#10MS);
	
	CASE _itemScheduler OF				
		0:	GetAxisStatus();
			_itemScheduler := 1;
						
		1:	GetPosition();
			_itemScheduler := 0;			
	END_CASE		
ELSE
	_pulseGenerator(IN := TRUE, PT := T#100MS);		
END_IF
END_METHOD

{attribute 'TcRpcEnable' := '1'}
METHOD MotorInit
VAR_INPUT
	Execute : BOOL;
END_VAR
VAR	
	cmd : STRING := 'INIT';
END_VAR
IF Execute THEN
	_logger.Information(_message.Reset().Append(_config.Name).Append(' - Enable the motor power stage').ToString());
	_serialCom.Send(Concat(cmd, AxesConst.AXIS_FILTER_WHEEL));	

	_cmdMotorInit := FALSE;	
END_IF
END_METHOD

{attribute 'TcRpcEnable' := '1'}
METHOD PROTECTED MoveAbsPosition 
VAR_INPUT
	Execute : BOOL;
	Position : LREAL;
END_VAR
VAR
	cmdSet : STRING := 'PSET';
	cmdGo : STRING := 'PGO';
	cmdCnt : STRING := '?CNT';
	cmd : STRING;	
END_VAR
IF Execute THEN

	_cmdMoveAbsPosition := TRUE;
	_posToDegree := Position;	
	
	IF _pulseMoveGenerator.Q THEN
		_pulseMoveGenerator(IN := FALSE, PT := T#10MS);
	
		CASE _itemMove OF
			0:	_logger.Information(_message.Reset().Append(_config.Name).Append(' - Move absolute position : ').
													 Append(TO_STRING(_posToDegree)).Append(' °').ToString());
								
				cmd := Concat(CONCAT(cmdSet, AxesConst.AXIS_FILTER_WHEEL), '=');				
				_serialCom.Send(CONCAT(cmd, LREAL_TO_STRING(_posToDegree * _convertDegreeToCount)));				
				_itemMove := 1;						
				
			1:  _serialCom.Send(Concat(cmdGo, AxesConst.AXIS_FILTER_WHEEL));											
				_itemMove := 2;	
				
			2:  _deliverMessages := EFeedbackMsgOwisPs10.CurrentPositionCounterMsg;	
				IF _currentPositionCounter <> (_posToDegree * _convertDegreeToCount) THEN					
					_serialCom.Send(Concat(cmdCnt, AxesConst.AXIS_FILTER_WHEEL));
					IsInMovingMsg := BOOL_TO_STRING(TRUE);	
				ELSE
					IsInMovingMsg := BOOL_TO_STRING(FALSE);	
					_itemMove := 3;	
				END_IF
								
			3: _cmdMoveAbsPosition := FALSE;
				_itemMove := 0;
			
		END_CASE			
	ELSE
		_pulseMoveGenerator(IN := TRUE, PT := T#100MS);	
	END_IF

END_IF
END_METHOD

METHOD PRIVATE ParseAxisStatus : STRING
VAR_INPUT
	CurrentAxisMode : STRING;
END_VAR
VAR
	Description : STRING;
END_VAR
IF CurrentAxisMode = 'I' THEN
	Description := 'Axis is not initialized';
ELSIF CurrentAxisMode = 'O' THEN
	Description := 'Axis is disabled';
ELSIF CurrentAxisMode = 'R' THEN
	Description := 'Axis initialized and ready';
ELSIF CurrentAxisMode = 'T' THEN
	Description := 'Axis is positioning in trapezoidal profile';
ELSIF CurrentAxisMode = 'V' THEN
	Description := 'Axis is operating in velocity mode';
ELSIF CurrentAxisMode = 'P' THEN
	Description := 'Reference motion is in progress';
ELSIF CurrentAxisMode = 'F' THEN
	Description := 'Axis is releasing a limit switch';
ELSIF CurrentAxisMode = 'L' THEN
	Description := 'Axis has been disabled after approaching a hardware limit switch(MINSTOP, MAXSTOP)';
ELSIF CurrentAxisMode = 'B' THEN
	Description := 'Aaxis has been stopped after approaching a brake switch(MINDEC, MAXDEC)';
ELSIF CurrentAxisMode = 'A' THEN
	Description := 'Axis has been disabled after limit switch error';
ELSIF CurrentAxisMode = 'M' THEN
	Description := 'Axis has been disabled after motion-controller error';
ELSIF CurrentAxisMode = 'Z' THEN
	Description := 'Axis has been disabled after timeout error';
ELSIF CurrentAxisMode = 'H' THEN
	Description := 'Phase initialization active (step motor axis)';
ELSIF CurrentAxisMode = 'U' THEN
	Description := 'Axis not enabled';
ELSIF CurrentAxisMode = 'E' THEN
	Description := 'Axis has been disabled after motion error';
ELSIF CurrentAxisMode = '?' THEN
	Description := 'Error, unknown state of axis';
ELSE
	Description := 'Unknown error';
END_IF

ParseAxisStatus := Description;
END_METHOD

{attribute 'TcRpcEnable' := '1'}
METHOD RaisePropertiesChanged
VAR_INPUT
	Execute : BOOL;
END_VAR
IF Execute THEN
	IF THIS^.Status <> TExecutionState.Ready THEN	
		_cmdRaiseProperties := FALSE;
		RETURN;
	END_IF	

	_cmdRaiseProperties := TRUE;
	
	IF _pulseGenerator.Q THEN
		_pulseGenerator(IN := FALSE, PT := T#10MS);	

		CASE _itemRaisedProperties OF
			0:  StateMsg := ' ';
				AxisStatusMsg := ' ';
				ErrMsg := ' ';
				PositionMsg := ' ';
				CustomMsg := ' ';
				
				_itemRaisedProperties := 10;
			
			10:  GetPosition();
				_itemRaisedProperties := 11;
			
			11:  GetAxisStatus();
				 _itemRaisedProperties := 12;
				 
			12:  ErrorMessages();
				 _itemRaisedProperties := 20;			
				 
			20:  _logger.Information(_message.Reset().Append(_config.Name).Append(' - PS10 Axis RaisePropertiesChanged').ToString());
				_cmdRaiseProperties := FALSE;				
				_itemRaisedProperties := 0;
			
		END_CASE
	ELSE
		_pulseGenerator(IN := TRUE, PT := T#100MS);	
	END_IF
END_IF
END_METHOD

{attribute 'TcRpcEnable' := '1'}
METHOD Reset
VAR_INPUT
	Execute : BOOL;
END_VAR
VAR
	cmd : STRING := 'RESETMB';
END_VAR
IF Execute THEN
	_logger.Information(_message.Reset().Append(_config.Name).Append(' - Release reset main board').ToString());
	_serialCom.Send(cmd);	
	
	_cmdReset := FALSE;
END_IF
END_METHOD

{attribute 'TcRpcEnable' := '1'}
METHOD SetDrivingCurrent
VAR_INPUT
	Execute : BOOL;
END_VAR
VAR
	cmdSet : STRING := 'DRICUR';
	cmd : STRING;
END_VAR
IF Execute THEN
	_logger.Information(_message.Reset().Append(_config.Name).Append(' - driving current with stepper motor: ').
		Append(TO_STRING(AxesConst.FW_DRIVING_CURRENT_IN_PERCENT)).ToString());
	
	cmd := Concat(CONCAT(cmdSet, AxesConst.AXIS_FILTER_WHEEL), '=');
	_serialCom.Send(CONCAT(cmd, TO_STRING(AxesConst.FW_DRIVING_CURRENT_IN_PERCENT)));	

	_cmdDrivingCurrent := FALSE;	
END_IF
END_METHOD

{attribute 'TcRpcEnable' := '1'}
METHOD SetHoldingCurrent
VAR_INPUT
	Execute : BOOL;
END_VAR
VAR
	cmdSet : STRING := 'HOLCUR';
	cmd : STRING;
END_VAR
IF Execute THEN
	_logger.Information(_message.Reset().Append(_config.Name).Append(' - holding current with stepper motor axes: ').
		Append(TO_STRING(AxesConst.FW_HOLDING_CURRENT_IN_PERCENT)).ToString());
	
	cmd := Concat(CONCAT(cmdSet, AxesConst.AXIS_FILTER_WHEEL), '=');
	_serialCom.Send(CONCAT(cmd, TO_STRING(AxesConst.FW_HOLDING_CURRENT_IN_PERCENT)));	

	_cmdHoldingCurrent := FALSE;	
END_IF
END_METHOD

{attribute 'TcRpcEnable' := '1'}
METHOD SetLimitSwitch
VAR_INPUT
	Execute : BOOL;
END_VAR
VAR
	cmdSet : STRING := 'SMK';
	cmd : STRING;
END_VAR
IF Execute THEN
	_logger.Information(_message.Reset().Append(_config.Name).Append(' -  limit switch mask for the axis: ').
		Append(TO_STRING(AxesConst.FW_LIMIT_SWITCH_MASK)).ToString());
	
	cmd := Concat(CONCAT(cmdSet, AxesConst.AXIS_FILTER_WHEEL), '=');
	_serialCom.Send(CONCAT(cmd, TO_STRING(AxesConst.FW_LIMIT_SWITCH_MASK)));	

	_cmdLimitSwitch := FALSE;	
END_IF
END_METHOD

{attribute 'TcRpcEnable' := '1'}
METHOD StopMotion
VAR_INPUT
	Execute : BOOL;
END_VAR
VAR
	cmd : STRING := 'STOP1';
END_VAR
IF Execute THEN	
	_logger.Information(_message.Reset().Append(_config.Name).Append(' - Stop motion').ToString());
	_serialCom.Send(cmd);
	
	_cmdStopMotion := FALSE;
END_IF
END_METHOD

END_FUNCTION_BLOCK

// ---- PMShared/Hardware/Devices/Lights/Evosens/EvosensLight.TcPOU
{attribute 'OPC.UA.DA' := '1'}
FUNCTION_BLOCK EvosensLight EXTENDS LightBase
VAR_INPUT
END_VAR
VAR_OUTPUT
END_VAR
VAR
	{attribute 'OPC.UA.DA' := '0'}
	_config : EvosensLightConfig;	
	{attribute 'OPC.UA.DA' := '0'}
	_coeAccess : CoeAccess;	
	{attribute 'OPC.UA.DA' := '0'}
	_initConfigSerialCom : BOOL;	
	{attribute 'OPC.UA.DA' := '0'}
	_suffix : STRING := Const.CR_LF;
	{attribute 'OPC.UA.DA' := '0'}
	_serialCom  : SerialCom(Prefix :='', Suffix := _suffix);
	{attribute 'OPC.UA.DA' := '0'}
	_refSerialCom : REFERENCE TO SerialCom(Prefix :='', Suffix := _suffix) := _serialCom;		 
	{attribute 'OPC.UA.DA' := '0'}
	_isReceived : BOOL;
	
	{attribute 'OPC.UA.DA' := '0'}
	_deliverMessages : INT;
		
	StatusMsg : STRING(255);
	SwitchOnMsg : STRING(255);
	PowerMsg : STRING(255);
	IntensityMsg : STRING(255);	
	TemperatureMsg : STRING(255);
	LightSourcesMsg : STRING(255);
	TimeLightSourceMsg  : STRING(255);
	CustomMsg : STRING(255);
		
	{region 'Commands'}
	
	{attribute 'OPC.UA.DA' := '0'}
	_setSwitchOnCmd : BOOL;
	{attribute 'OPC.UA.DA' := '0'}
	_getSwitchOnCmd : BOOL;
	{attribute 'OPC.UA.DA' := '0'}
	_setPowerCmd : BOOL;
	{attribute 'OPC.UA.DA' := '0'}
	_getPowerCmd : BOOL;
	{attribute 'OPC.UA.DA' := '0'}
	_setIntensityCmd : BOOL;
	{attribute 'OPC.UA.DA' := '0'}
	_getIntensityCmd : BOOL;
	{attribute 'OPC.UA.DA' := '0'}
	_getTimeLightSourceCmd : BOOL;
	{attribute 'OPC.UA.DA' := '0'}
	_getLightSourcesCmd : BOOL;
	{attribute 'OPC.UA.DA' := '0'}
	_customCmd : BOOL;
	{attribute 'OPC.UA.DA' := '0'}			  		   
	_raisePropertiesCmd : BOOL;
	
	{attribute 'OPC.UA.DA' := '0'}
	_lightId : UINT; 
	{attribute 'OPC.UA.DA' := '0'}
	_switchOn : BOOL;
	{attribute 'OPC.UA.DA' := '0'}
	_setPower : LREAL;
	{attribute 'OPC.UA.DA' := '0'}
	_setIntensity : LREAL;
	{attribute 'OPC.UA.DA' := '0'}
	_cmd : STRING;	
		 
	{endregion}			
	
	{attribute 'OPC.UA.DA' := '0'}
	_initDevice : BOOL;	
	 
	{attribute 'OPC.UA.DA' := '0'}
	_lightSources : ARRAY [0..Const.PHOTOLUM_NUMBER_LIGHT_SOURCE] OF STRING(255);  
	
	{attribute 'OPC.UA.DA' := '0'}
	_itemScheduler : INT;
	{attribute 'OPC.UA.DA' := '0'}
	_itemInitScheduler : INT;
	{attribute 'OPC.UA.DA' := '0'}
	_itemExecScheduler : INT;		
	{attribute 'OPC.UA.DA' := '0'}
	_itemRaisedProperties : INT;			
	{attribute 'OPC.UA.DA' := '0'}
	_pulseGenerator : TON;	
	{attribute 'OPC.UA.DA' := '0'}
	_initPulseGenerator : TON;	
	{attribute 'OPC.UA.DA' := '0'}	
	_execPulseGenerator : TON;	
	
	{attribute 'OPC.UA.DA' := '0'}
	message : STRING;
	{attribute 'OPC.UA.DA' := '0'}
	lastMessage : STRING;	
	{attribute 'OPC.UA.DA' := '0'}
	sSubStr4 : STRING(4) := '';			
	{attribute 'OPC.UA.DA' := '0'}
	stringLength : INT;
	{attribute 'OPC.UA.DA' := '0'}
	_numberOfElements : DINT;
	{attribute 'OPC.UA.DA' := '0'}
	_indexNumberOfElements : INT;
END_VAR

IF NOT InitConfigSerialCom THEN
	ConfigureSerialCom();
ELSIF THIS^.Status = TExecutionState.Ready THEN
	SUPER^();	

	IF _refSerialCom.ErrorReceiveId = COMERROR_NOERROR THEN
		_refSerialCom(TxBuffer:= HardwareGlobalVariables.TxBufferLight, 
		 	      	  RxBuffer:= HardwareGlobalVariables.RxBufferLight);
	END_IF				  
	
	// Init device
	InitDevice(); 				  				 	
	
	IF StateMsg <> ANY_TO_STRING(State) THEN
		StateMsg := ANY_TO_STRING(State);
	END_IF
	
	// Deliver messages
	IF _refSerialCom.IsReceived THEN	
		lastMessage := _refSerialCom.LastReceivedString;			
		stringLength := LEN(lastMessage);
		
		IF stringLength > 2 THEN
			message := LEFT(lastMessage, stringLength - 2);
		ELSE
			message := ' ';
		END_IF; 	
			
		CASE _deliverMessages OF			
			EFeedbackMsgArduinoLight.SwitchOnMsg :
				SwitchOnMsg := message;	
			EFeedbackMsgArduinoLight.PowerMsg :
				PowerMsg := message;	
			EFeedbackMsgArduinoLight.IntensityMsg :
				IntensityMsg := message;	
			EFeedbackMsgArduinoLight.TemperatureMsg :
				TemperatureMsg := message;	
			EFeedbackMsgArduinoLight.LightSourcesMsg :
				LightSourcesMsg := message;			
				_logger.Information(_message.Reset().Append('LightSourcesMsg: ').Append(LightSourcesMsg).ToString());	
			EFeedbackMsgArduinoLight.TimeLightSourceMsg :
				TimeLightSourceMsg := message;	
			EFeedbackMsgArduinoLight.CustomMsg :
				CustomMsg := message;	
		END_CASE
	
		_deliverMessages := 0;
	END_IF								   							   	
		
	SetSwitchOn(_setSwitchOnCmd, TO_STRING(_lightId), _switchOn); 
	GetSwitchOn(_getSwitchOnCmd, TO_STRING(_lightId));
	SetPower(_setPowerCmd, TO_STRING(_lightId), _setPower);
	GetPower(_getPowerCmd, TO_STRING(_lightId));
	//SetIntensity(_setIntensityCmd, TO_STRING(_lightId), _setIntensity);
	//GetIntensity(_getIntensityCmd, TO_STRING(_lightId));
	GetTimeLightSource(_getTimeLightSourceCmd, TO_STRING(_lightId));
	GetLightSources(_getLightSourcesCmd);
	CustomCommand(_customCmd, _cmd);
	RaisePropertiesChanged(_raisePropertiesCmd, TO_STRING(_lightId));
	
	IF _initDevice AND NOT _setSwitchOnCmd AND NOT _getSwitchOnCmd AND NOT _setPowerCmd AND NOT _getPowerCmd AND NOT _setIntensityCmd AND NOT _getIntensityCmd
	   AND NOT _getTimeLightSourceCmd AND NOT _getLightSourcesCmd AND NOT _customCmd AND NOT _raisePropertiesCmd THEN
		MessageScheduler();
	END_IF
END_IF

METHOD ConfigureSerialCom
VAR_INPUT
END_VAR
IF _coeAccess.CoeOperation.Ready THEN
	_logger.Information(_message.Reset().Append('Start configuration com serial').ToString());
END_IF;	

_coeAccess.CoeOperation.Start();
_coeAccess(SerialCommunication := _config.SerialCommunication);
	
IF _coeAccess.CoeOperation.Done THEN
	_coeAccess.SetDone();	
	
	_Logger.Information(_message.Reset().
							Append('{').Append(TO_STRING(THIS^.Family)).Append('} : ').
							Append(' - Status : ').Append(TO_STRING(_coeAccess.Status)).ToString());	
	InitConfigSerialCom := TRUE;
END_IF
 
IF _coeAccess.CoeOperation.Error THEN	
	_coeAccess.SetError(0);
	
	_Logger.Error(_message.Reset().
							Append('{').Append(TO_STRING(THIS^.Family)).Append('} : ').
							Append(' - Status : ').Append(TO_STRING(_coeAccess.Status)).ToString());
	InitConfigSerialCom := TRUE;
END_IF

THIS^.Status := _coeAccess.Status;
State := _coeAccess.Status;
END_METHOD

{attribute 'TcRpcEnable' := '1'}
(** Custom command **)
METHOD CustomCommand
VAR_INPUT
	Execute : BOOL;
	Cmd : STRING;
END_VAR
IF Execute THEN
	_logger.Information(_message.Reset().Append(_config.Name).Append(' - Custom command : ').Append(Cmd).ToString());	
	_deliverMessages := EFeedbackMsgArduinoLight.CustomMsg;														
	_serialCom.Send(Cmd);	
	_customCmd := FALSE;
END_IF
END_METHOD

METHOD FB_init : BOOL
VAR_INPUT
	bInitRetains : BOOL; // if TRUE, the retain variables are initialized (warm start / cold start)
	bInCopyCode : BOOL;  // if TRUE, the instance afterwards gets moved into the copy code (online change)
	Config : EvosensLightConfig;
END_VAR
IF Config.IsEnabled THEN
	_config := Config;
	
	SUPER^._lightConfig.Name := Config.Name;
	SUPER^._lightConfig.DeviceID := Config.DeviceID;
	SUPER^._lightConfig.IsEnabled := Config.IsEnabled;
	SUPER^._lightConfig.LogLevel := Config.LogLevel;
	
	SUPER^.Name := Config.Name;
	SUPER^.DeviceID := Config.DeviceID;	
	THIS^.Family := DeviceFamily.Light;
		
	_Logger.Information(_message.Reset().Append('Init ').
							Append('{').Append(TO_STRING(THIS^.Family)).Append('} - ').
							Append('{').Append(TO_STRING(Config.Name)).Append('}').ToString());																													
END_IF
END_METHOD

{attribute 'TcRpcEnable' := '1'}
METHOD GetIntensity
VAR_INPUT
	Execute : BOOL;
	LightId : STRING;
END_VAR
VAR
	cmd : STRING := '*amps ';
END_VAR
IF Execute THEN	
	_deliverMessages := EFeedbackMsgArduinoLight.IntensityMsg;
	_serialCom.Send(CONCAT(cmd, LightId));
	
	_getIntensityCmd := FALSE;
END_IF
END_METHOD

METHOD GetLightSources
VAR_INPUT
	Execute: BOOL;
END_VAR
VAR
	cmd : STRING := '*light';
END_VAR
IF Execute THEN
	_logger.Information(_message.Reset().Append(_config.Name).Append(' - GetLightSources').ToString());
	_deliverMessages := EFeedbackMsgArduinoLight.LightSourcesMsg;
	_serialCom.Send(cmd);	
	
	_getLightSourcesCmd := FALSE;
END_IF
END_METHOD

{attribute 'TcRpcEnable' := '1'}
METHOD GetPower
VAR_INPUT
	Execute : BOOL;
	LightId : STRING;
END_VAR
VAR
	cmd : STRING := '*power ';
END_VAR
IF Execute THEN	
	_deliverMessages := EFeedbackMsgArduinoLight.PowerMsg;
	_serialCom.Send(CONCAT(cmd, LightId));
	
	 _getPowerCmd := FALSE;
END_IF
END_METHOD

{attribute 'TcRpcEnable' := '1'}
METHOD GetSwitchOn
VAR_INPUT
	Execute : BOOL;
	LightId : STRING;
END_VAR
VAR
	cmd : STRING := '*switch ';
END_VAR
IF Execute THEN	
	_deliverMessages := EFeedbackMsgArduinoLight.SwitchOnMsg;
	_serialCom.Send(CONCAT(cmd, LightId));
				
	_getSwitchOnCmd := FALSE;	
END_IF
END_METHOD

METHOD GetTemperature
VAR_INPUT
	LightId : STRING;
END_VAR
VAR
	cmd : STRING := '*temp ';
END_VAR
_deliverMessages := EFeedbackMsgArduinoLight.TemperatureMsg;
_serialCom.Send(CONCAT(cmd, LightId));
END_METHOD

METHOD GetTimeLightSource
VAR_INPUT
	Execute: BOOL;
	LightId : STRING;
END_VAR
VAR
	cmd : STRING := '*time ';
END_VAR
IF Execute THEN
	_logger.Information(_message.Reset().Append(_config.Name).Append(' - GetTimeLightSource - ').Append(LightId).ToString());
	_deliverMessages := EFeedbackMsgArduinoLight.TimeLightSourceMsg;
	_serialCom.Send(CONCAT(cmd, LightId));	
	
	_getTimeLightSourceCmd := FALSE;
END_IF
END_METHOD

PROPERTY InitConfigSerialCom : BOOL
GET
InitConfigSerialCom := _initConfigSerialCom;
END_GET
SET
_initConfigSerialCom := InitConfigSerialCom;
END_SET
END_PROPERTY

METHOD InitDevice
VAR_INPUT
END_VAR
VAR
	numElements : INT := 0;
    commaPos : INT;
    tempStr : STRING; 
	Separator : STRING := ',';
END_VAR
IF NOT _initDevice THEN	
	IF _initPulseGenerator.Q THEN
		_initPulseGenerator(IN := FALSE, PT := T#10MS);
			
		CASE _itemInitScheduler OF					
			0:	_logger.Information(_message.Reset().Append(_config.Name).Append(' - Init device').ToString());
				//_getLightSourcesCmd := TRUE;
				_itemInitScheduler := 50;
			
			1:	IF LightSourcesMsg <> '' THEN				
					tempStr := LightSourcesMsg;
					WHILE (LEN(tempStr) > 0) DO
						commaPos := FIND(tempStr, Separator);
						IF commaPos > 0 THEN
							_lightSources[numElements] := LEFT(tempStr, commaPos - 1);						
							tempStr := RIGHT(tempStr, LEN(tempStr) - commaPos);
						ELSE
							_lightSources[numElements] := tempStr;
							tempStr := ''; 
						END_IF
						_logger.Information(_message.Reset().Append(_config.Name).Append(' - ').Append(TO_STRING(numElements)).Append(': ').Append(_lightSources[numElements]).ToString());
						numElements := numElements + 1;						
					END_WHILE
														
					IF (numElements - 1) <> 0 THEN
						_numberOfElements := numElements;
						//_itemInitScheduler := 10; GVA
						_itemInitScheduler := 50;
					ELSE
						_itemInitScheduler := 40;	
					END_IF				
					
					_deliverMessages := -1;
				END_IF
			
			10: IF (_indexNumberOfElements >= 0) AND (_indexNumberOfElements < _numberOfElements) THEN
					tempStr := CONCAT(_lightSources[_indexNumberOfElements], ' 0');
					_serialCom.Send(CONCAT('*power ', tempStr));				
					_logger.Information(_message.Reset().Append(_config.Name).Append(' - ').Append(_lightSources[_indexNumberOfElements]).Append(' - Power: 0').ToString());	
					_indexNumberOfElements := _indexNumberOfElements + 1;
					
				ELSE
					_indexNumberOfElements := 0;
					_itemInitScheduler := 11;					
				END_IF	
			
			11: IF (_indexNumberOfElements >= 0) AND (_indexNumberOfElements < _numberOfElements) THEN
					tempStr := CONCAT(_lightSources[_indexNumberOfElements], ' 1');
					_serialCom.Send(CONCAT('*swit ', tempStr));
					_logger.Information(_message.Reset().Append(_config.Name).Append(' - ').Append(_lightSources[_indexNumberOfElements]).Append(' - Switch ON').ToString());
					_indexNumberOfElements := _indexNumberOfElements + 1;					
				ELSE
					_indexNumberOfElements := 0;
					_itemInitScheduler := 50;
				END_IF	

			41: _logger.Error(_message.Reset().Append(_config.Name).Append(' - numElements is empty: ').ToString());
				_itemInitScheduler := 50;	
		
			50: _initDevice := TRUE;
				_itemInitScheduler := 0;	
				_logger.Information(_message.Reset().Append(_config.Name).Append(' - Init device done').ToString());	
		END_CASE
	ELSE
		_initPulseGenerator(IN := TRUE, PT := T#100MS);		
	END_IF	
END_IF
END_METHOD

METHOD MessageScheduler
VAR_INPUT
END_VAR
VAR
	
END_VAR
IF _pulseGenerator.Q THEN
	_pulseGenerator(IN := FALSE, PT := T#10MS);
		
	CASE _itemScheduler OF					
		0:	_getSwitchOnCmd := TRUE;
			_itemScheduler := 1;
			
		1:	_getPowerCmd := TRUE;
			_itemScheduler := 2;
			
		2:  //GetTemperature(_lightID);			
			_itemScheduler := 10;
			
		10: IF _lightId > 0 AND _lightId < Const.PHOTOLUM_NUMBER_LIGHT_SOURCE THEN
				_lightId := _lightId + 1;				
			ELSE
				_lightId := 1;
			END_IF
			
			
			_itemScheduler := 0;
									
	END_CASE
ELSE
	_pulseGenerator(IN := TRUE, PT := T#250MS);		
END_IF


IF _pulseIsAliveGenerator.Q THEN
	_pulseIsAliveGenerator(IN := FALSE, PT := T#10MS);
		
	IsAlive();	
ELSE
	_pulseIsAliveGenerator(IN := TRUE, PT := T#1000MS);		
END_IF
END_METHOD

{attribute 'TcRpcEnable' := '1'}
METHOD RaisePropertiesChanged
VAR_INPUT
	Execute : BOOL;
	LightId : STRING;
END_VAR
VAR
	numElements : INT := 0;
    commaPos : INT;
    tempStr : STRING; 
	Separator : STRING := ',';
END_VAR
IF Execute THEN
	_raisePropertiesCmd := TRUE;
	IF LightId <> '' THEN
		_lightId := STRING_TO_UINT(LightId);
	END_IF
	
	IF _pulseGenerator.Q THEN
		_pulseGenerator(IN := FALSE, PT := T#10MS);	

		CASE _itemRaisedProperties OF
			0:  SwitchOnMsg := ' ';
				PowerMsg := ' ';		
				IntensityMsg := ' ';
				LightSourcesMsg := ' ';		
				TimeLightSourceMsg := ' ';		
				_itemRaisedProperties := 1;					

			1:  IF _lightId > 0 AND _lightId <= Const.PHOTOLUM_NUMBER_LIGHT_SOURCE THEN
					_itemRaisedProperties := 50;	
				ELSE
					_itemRaisedProperties := 40;	
				END_IF  
				
			10: _getSwitchOnCmd := TRUE;													
				_itemRaisedProperties := 11;
				
			11: IF SwitchOnMsg <> ' ' THEN
					_itemRaisedProperties := 12;
				END_IF	
				
			12: _getPowerCmd := TRUE;													
				_itemRaisedProperties := 13;
				
			13: IF PowerMsg <> ' ' THEN
					_itemRaisedProperties := 16;
				END_IF
							
			16: _getTimeLightSourceCmd := TRUE;													
				_itemRaisedProperties := 17;
				
			17: IF TimeLightSourceMsg <> ' ' THEN
					_itemRaisedProperties := 50;
				END_IF
			
			40: _logger.Error(_message.Reset().Append(_config.Name).Append(' - RaisePropertiesChanged - LightId is empty').ToString());
				_itemRaisedProperties := 50;
			
			50:  _logger.Information(_message.Reset().Append(_config.Name).Append(' - RaisePropertiesChanged').ToString());
				_raisePropertiesCmd := FALSE;				
				_itemRaisedProperties := 0;
			
		END_CASE
	ELSE
		_pulseGenerator(IN := TRUE, PT := T#100MS);	
	END_IF
END_IF
END_METHOD

{attribute 'TcRpcEnable' := '1'}
METHOD SetIntensity
VAR_INPUT
	Execute : BOOL;
	LightId : STRING;
	Intensity : LREAL;
END_VAR
VAR
	cmd : STRING := '*amps ';
	tmpConcatLightIdIntensity : STRING;
END_VAR
IF Execute THEN	
	_setIntensityCmd := TRUE;
	_setIntensity := Intensity; 
	IF LightId <> '' THEN
		_lightId := STRING_TO_UINT(LightId);
	END_IF
	
	IF _execPulseGenerator.Q THEN
		_execPulseGenerator(IN := FALSE, PT := T#10MS);
			
		CASE _itemExecScheduler OF
			0:  IF _lightId > 0 AND _lightId <= Const.PHOTOLUM_NUMBER_LIGHT_SOURCE THEN
					_itemExecScheduler := 10;	
				ELSE
					_itemExecScheduler := 40;	
				END_IF
				
				_deliverMessages := -1;

			10: tmpConcatLightIdIntensity := CONCAT(CONCAT(TO_STRING(_lightId), ' '), TO_STRING(Intensity));

				_logger.Information(_message.Reset().Append(_config.Name).Append(' - ').Append(TO_STRING(_lightId)).Append(' - SetIntensity : ').Append(TO_STRING(_lightId)).Append(' - ').Append(TO_STRING(Intensity)).ToString());
				_serialCom.Send(CONCAT(cmd, TO_STRING(tmpConcatLightIdIntensity)));
				_itemExecScheduler := 11;
			
			11:  _getIntensityCmd := TRUE;
				_itemExecScheduler := 50;
			
			40: _logger.Error(_message.Reset().Append(_config.Name).Append(' - SetIntensity - light id is not valid').ToString());
				_itemExecScheduler := 50;
		
			50:  _setIntensityCmd := FALSE;	
				_itemExecScheduler := 0;		
								
		END_CASE
	ELSE
		_execPulseGenerator(IN := TRUE, PT := T#100MS);	
	END_IF
END_IF
END_METHOD

{attribute 'TcRpcEnable' := '1'}
METHOD SetPower
VAR_INPUT
	Execute : BOOL;
	LightId : STRING;
	Power : LREAL;
END_VAR
VAR
	cmd : STRING := '*power ';
	tmpConcatLightIdPower : STRING;
END_VAR
IF Execute THEN	
	_setPowerCmd := TRUE;		
	_setPower := Power;	
	IF LightId <> '' THEN
		_lightId := STRING_TO_UINT(LightId);
	END_IF
	
	IF _execPulseGenerator.Q THEN
		_execPulseGenerator(IN := FALSE, PT := T#10MS);
			
		CASE _itemExecScheduler OF
			0: IF _lightId > 0 AND _lightId <= Const.PHOTOLUM_NUMBER_LIGHT_SOURCE THEN
					_itemExecScheduler := 10;	
				ELSE
					_itemExecScheduler := 40;	
				END_IF
				
				_deliverMessages := -1;

			10: tmpConcatLightIdPower := CONCAT(CONCAT(TO_STRING(_lightId), ' '), TO_STRING(Power));

				_logger.Information(_message.Reset().Append(_config.Name).Append(' - ').Append(TO_STRING(_lightId)).Append(' - SetPower : ').Append(TO_STRING(Power)).ToString());
				_serialCom.Send(CONCAT(cmd, TO_STRING(tmpConcatLightIdPower)));
				_itemExecScheduler := 11;
			
			11:  _getPowerCmd := TRUE;
				_itemExecScheduler := 50;
			
			40: _logger.Error(_message.Reset().Append(_config.Name).Append(' - SetPower - light id is not valid').ToString());
				_itemExecScheduler := 50;
	
			50:  _setPowerCmd := FALSE;	
				_itemExecScheduler := 0;		
								
		END_CASE
	ELSE
		_execPulseGenerator(IN := TRUE, PT := T#100MS);	
	END_IF
END_IF
END_METHOD

{attribute 'TcRpcEnable' := '1'}
METHOD SetSwitchOn
VAR_INPUT
	Execute : BOOL;	
	LightId : STRING;
	SwitchOn : BOOL;
END_VAR
VAR
	cmd : STRING := '*switch ';
	tmpConcatLightIdSwitchOn : STRING;
	tmp : STRING;
	switchOnValue : STRING;
END_VAR
IF Execute THEN	
	_setSwitchOnCmd := TRUE;	
	_switchOn := SwitchOn; 
	
	IF LightId <> '' THEN
		_lightId := STRING_TO_UINT(LightId);
	END_IF	
	
	IF _execPulseGenerator.Q THEN
		_execPulseGenerator(IN := FALSE, PT := T#10MS);
			
		CASE _itemExecScheduler OF
			0:  IF _lightId > 0 AND _lightId <= Const.PHOTOLUM_NUMBER_LIGHT_SOURCE THEN
					_itemExecScheduler := 10;	
				ELSE
					_itemExecScheduler := 40;	
				END_IF
				
				_deliverMessages := -1;

			10:	IF _switchOn THEN
					switchOnValue := 'ON';
				ELSE
					switchOnValue := 'OFF';
				END_IF
				tmpConcatLightIdSwitchOn := CONCAT(CONCAT(TO_STRING(_lightId), ' '), TO_STRING(switchOnValue));
				
				_logger.Information(_message.Reset().Append(_config.Name).Append(' - ').Append(TO_STRING(_lightId)).Append(' - SwitchOn : ').Append(TO_STRING(switchOnValue)).ToString());
				tmp := CONCAT(cmd, TO_STRING(tmpConcatLightIdSwitchOn));
				_serialCom.Send(tmp);
				_itemExecScheduler := 11;
			
			11:  _getSwitchOnCmd := TRUE;
				_itemExecScheduler := 50;
				
			40: _logger.Error(_message.Reset().Append(_config.Name).Append(' - SwitchOn - light id is not valid').ToString());
				_itemExecScheduler := 50;
				
			50:  _setSwitchOnCmd := FALSE;	
				_switchOn := FALSE;
				_itemExecScheduler := 0;		
								
		END_CASE
	ELSE
		_execPulseGenerator(IN := TRUE, PT := T#200MS);	
	END_IF
END_IF
END_METHOD

END_FUNCTION_BLOCK

// ---- PMShared/Hardware/Devices/Lights/LightBase.TcPOU
FUNCTION_BLOCK ABSTRACT LightBase EXTENDS TExecution IMPLEMENTS IDevice
VAR_INPUT
END_VAR
VAR_OUTPUT
END_VAR
VAR
	{attribute 'OPC.UA.DA' := '0'}
	_name : STRING;
	{attribute 'OPC.UA.DA' := '0'}
	_deviceID : STRING;				
	{attribute 'OPC.UA.DA' := '0'}	
	_family : DeviceFamily;	
	{attribute 'OPC.UA.DA' := '0'}
	_logger : Logger;
	{attribute 'OPC.UA.DA' := '0'}
	_message : StringBuilder;
	{attribute 'OPC.UA.DA' := '0'}
	_lightConfig : DeviceConfiguration;	
	
	{attribute 'OPC.UA.DA' := '0'}
	_lifeTimeCount : UINT;
	{attribute 'OPC.UA.DA' := '0'}
	_notifyIsAlive : BOOL;
	{attribute 'OPC.UA.DA' := '0'}
	_pulseIsAliveGenerator : TON;				
		
	StateMsg : STRING(255);
	IsAliveMsg : STRING(255);
END_VAR

// Check if it's still alive	
IF _notifyIsAlive THEN
	IsAliveMsg := TO_STRING(_lifeTimeCount);
	_notifyIsAlive := FALSE;
END_IF

IF HardwareGlobalVariables.LightState <> State THEN
	HardwareGlobalVariables.LightState := State;
	StateMsg := ANY_TO_STRING(State);		
END_IF

MessageSchedulerBase();

PROPERTY DeviceID : STRING
GET
DeviceID := _deviceID;
END_GET
SET
_deviceID := DeviceID;
END_SET
END_PROPERTY

PROPERTY Family : DeviceFamily
GET
Family := _family;
END_GET
SET
_family := Family;
END_SET
END_PROPERTY

METHOD IsAlive
VAR_INPUT
END_VAR
_notifyIsAlive := TRUE;

IF _lifeTimeCount < 5 THEN
	_lifeTimeCount := _lifeTimeCount + 1;
ELSE
	_lifeTimeCount := 1;
END_IF
END_METHOD

METHOD MessageSchedulerBase
VAR_INPUT
END_VAR
IF _pulseIsAliveGenerator.Q THEN
	_pulseIsAliveGenerator(IN := FALSE, PT := T#10MS);
		
	IsAlive();	
ELSE
	_pulseIsAliveGenerator(IN := TRUE, PT := T#1000MS);		
END_IF
END_METHOD

PROPERTY Name : STRING
GET
Name := _name;
END_GET
SET
_name := Name;
END_SET
END_PROPERTY

METHOD ABSTRACT SetIntensity
VAR_INPUT
	Execute : BOOL;
	LightId : STRING;
	Intensity : LREAL;
END_VAR
END_METHOD

END_FUNCTION_BLOCK

// ---- PMShared/Hardware/Devices/Lights/Arduino/ArduinoLight.TcPOU
{attribute 'OPC.UA.DA' := '1'}
FUNCTION_BLOCK ArduinoLight EXTENDS LightBase
VAR_INPUT
END_VAR
VAR_OUTPUT
END_VAR
VAR
	{attribute 'OPC.UA.DA' := '0'}
	_config : ArduinoLightConfig;	
	{attribute 'OPC.UA.DA' := '0'}
	_coeAccess : CoeAccess;	
	{attribute 'OPC.UA.DA' := '0'}
	_initConfigSerialCom : BOOL;	
	{attribute 'OPC.UA.DA' := '0'}
	_suffix : STRING := Const.CR_LF;
	{attribute 'OPC.UA.DA' := '0'}
	_serialCom  : SerialCom(Prefix :='', Suffix := _suffix);
	{attribute 'OPC.UA.DA' := '0'}
	_refSerialCom : REFERENCE TO SerialCom(Prefix :='', Suffix := _suffix) := _serialCom;		 
	{attribute 'OPC.UA.DA' := '0'}
	_isReceived : BOOL;
	
	{attribute 'OPC.UA.DA' := '0'}
	_deliverMessages : INT;
		
	StatusMsg : STRING(255);
	SwitchOnMsg : STRING(255);
	PowerMsg : STRING(255);
	IntensityMsg : STRING(255);	
	TemperatureMsg : STRING(255);
	LightSourcesMsg : STRING(255);
	TimeLightSourceMsg  : STRING(255);
	CustomMsg : STRING(255);
		
	{region 'Commands'}
	
	{attribute 'OPC.UA.DA' := '0'}
	_setSwitchOnCmd : BOOL;
	{attribute 'OPC.UA.DA' := '0'}
	_getSwitchOnCmd : BOOL;
	{attribute 'OPC.UA.DA' := '0'}
	_setPowerCmd : BOOL;
	{attribute 'OPC.UA.DA' := '0'}
	_getPowerCmd : BOOL;
	{attribute 'OPC.UA.DA' := '0'}
	_setIntensityCmd : BOOL;
	{attribute 'OPC.UA.DA' := '0'}
	_getIntensityCmd : BOOL;
	{attribute 'OPC.UA.DA' := '0'}
	_getTimeLightSourceCmd : BOOL;
	{attribute 'OPC.UA.DA' := '0'}
	_getLightSourcesCmd : BOOL;
	{attribute 'OPC.UA.DA' := '0'}
	_customCmd : BOOL;
	{attribute 'OPC.UA.DA' := '0'}			  		   
	_raisePropertiesCmd : BOOL;
	
	{attribute 'OPC.UA.DA' := '0'}
	_lightId : STRING; 
	{attribute 'OPC.UA.DA' := '0'}
	_switchOn : BOOL;
	{attribute 'OPC.UA.DA' := '0'}
	_setPower : LREAL;
	{attribute 'OPC.UA.DA' := '0'}
	_setIntensity : LREAL;
	{attribute 'OPC.UA.DA' := '0'}
	_cmd : STRING;	
		 
	{endregion}			
	
	{attribute 'OPC.UA.DA' := '0'}
	_initDevice : BOOL;	
	 
	{attribute 'OPC.UA.DA' := '0'}
	_lightSources : ARRAY [0..Const.PHOTOLUM_NUMBER_LIGHT_SOURCE] OF STRING(255);  
	
	{attribute 'OPC.UA.DA' := '0'}
	_itemScheduler : INT;
	{attribute 'OPC.UA.DA' := '0'}
	_itemInitScheduler : INT;
	{attribute 'OPC.UA.DA' := '0'}
	_itemExecScheduler : INT;		
	{attribute 'OPC.UA.DA' := '0'}
	_itemRaisedProperties : INT;			
	{attribute 'OPC.UA.DA' := '0'}
	_pulseGenerator : TON;	
	{attribute 'OPC.UA.DA' := '0'}
	_initPulseGenerator : TON;	
	{attribute 'OPC.UA.DA' := '0'}	
	_execPulseGenerator : TON;	
	
	{attribute 'OPC.UA.DA' := '0'}
	message : STRING;
	{attribute 'OPC.UA.DA' := '0'}
	lastMessage : STRING;	
	{attribute 'OPC.UA.DA' := '0'}
	sSubStr4 : STRING(4) := '';			
	{attribute 'OPC.UA.DA' := '0'}
	stringLength : INT;
	{attribute 'OPC.UA.DA' := '0'}
	_numberOfElements : DINT;
	{attribute 'OPC.UA.DA' := '0'}
	_indexNumberOfElements : INT;
END_VAR

IF NOT InitConfigSerialCom THEN
	ConfigureSerialCom();
ELSIF THIS^.Status = TExecutionState.Ready THEN
	SUPER^();	

	IF _refSerialCom.ErrorReceiveId = COMERROR_NOERROR THEN
		_refSerialCom(TxBuffer:= HardwareGlobalVariables.TxBufferLight, 
		 	      	  RxBuffer:= HardwareGlobalVariables.RxBufferLight);
	END_IF				  
	
	// Init device
	InitDevice();		  				 
	
	IF StateMsg <> ANY_TO_STRING(State) THEN
		StateMsg := ANY_TO_STRING(State);
	END_IF
	
	// Deliver messages
	IF _refSerialCom.IsReceived THEN	
		lastMessage := _refSerialCom.LastReceivedString;			
		stringLength := LEN(lastMessage);
		
		IF stringLength > 2 THEN
			message := LEFT(lastMessage, stringLength - 2);
		ELSE
			message := ' ';
		END_IF; 	
			
		CASE _deliverMessages OF			
			EFeedbackMsgArduinoLight.SwitchOnMsg :
				SwitchOnMsg := message;	
			EFeedbackMsgArduinoLight.PowerMsg :
				PowerMsg := message;	
			EFeedbackMsgArduinoLight.IntensityMsg :
				IntensityMsg := message;	
			EFeedbackMsgArduinoLight.TemperatureMsg :
				TemperatureMsg := message;	
			EFeedbackMsgArduinoLight.LightSourcesMsg :
				LightSourcesMsg := message;			
				_logger.Information(_message.Reset().Append('LightSourcesMsg: ').Append(LightSourcesMsg).ToString());	
			EFeedbackMsgArduinoLight.TimeLightSourceMsg :
				TimeLightSourceMsg := message;	
			EFeedbackMsgArduinoLight.CustomMsg :
				CustomMsg := message;	
		END_CASE
		
		_deliverMessages := 0;
	END_IF								   							   	
		
	SetSwitchOn(_setSwitchOnCmd, _lightId, _switchOn); 
	GetSwitchOn(_getSwitchOnCmd, _lightId);
	SetPower(_setPowerCmd, _lightId, _setPower);
	GetPower(_getPowerCmd, _lightId);
	SetIntensity(_setIntensityCmd, _lightId, _setIntensity);
	GetIntensity(_getIntensityCmd, _lightId);
	GetTimeLightSource(_getTimeLightSourceCmd, _lightId);
	GetLightSources(_getLightSourcesCmd);
	CustomCommand(_customCmd, _cmd);
	RaisePropertiesChanged(_raisePropertiesCmd, _lightId);
	
	IF _initDevice AND NOT _setSwitchOnCmd AND NOT _getSwitchOnCmd AND NOT _setPowerCmd AND NOT _getPowerCmd AND NOT _setIntensityCmd AND NOT _getIntensityCmd
	   AND NOT _getTimeLightSourceCmd AND NOT _getLightSourcesCmd AND NOT _customCmd AND NOT _raisePropertiesCmd THEN
		MessageScheduler();
	END_IF
END_IF

METHOD ConfigureSerialCom
VAR_INPUT
END_VAR
IF _coeAccess.CoeOperation.Ready THEN
	_logger.Information(_message.Reset().Append('Start configuration com serial').ToString());
END_IF;	

_coeAccess.CoeOperation.Start();
_coeAccess(SerialCommunication := _config.SerialCommunication);
	
IF _coeAccess.CoeOperation.Done THEN
	_coeAccess.SetDone();	
	
	_Logger.Information(_message.Reset().
							Append('{').Append(TO_STRING(THIS^.Family)).Append('} : ').
							Append(' - Status : ').Append(TO_STRING(_coeAccess.Status)).ToString());	
	InitConfigSerialCom := TRUE;
END_IF
 
IF _coeAccess.CoeOperation.Error THEN	
	_coeAccess.SetError(0);
	
	_Logger.Error(_message.Reset().
							Append('{').Append(TO_STRING(THIS^.Family)).Append('} : ').
							Append(' - Status : ').Append(TO_STRING(_coeAccess.Status)).ToString());
	InitConfigSerialCom := TRUE;
END_IF

THIS^.Status := _coeAccess.Status;
State := _coeAccess.Status;
END_METHOD

{attribute 'TcRpcEnable' := '1'}
(** Custom command **)
METHOD CustomCommand
VAR_INPUT
	Execute : BOOL;
	Cmd : STRING;
END_VAR
IF Execute THEN
	_logger.Information(_message.Reset().Append(_config.Name).Append(' - Custom command : ').Append(Cmd).ToString());	
	_deliverMessages := EFeedbackMsgArduinoLight.CustomMsg;														
	_serialCom.Send(Cmd);	
	_customCmd := FALSE;
END_IF
END_METHOD

METHOD FB_init : BOOL
VAR_INPUT
	bInitRetains : BOOL; // if TRUE, the retain variables are initialized (warm start / cold start)
	bInCopyCode : BOOL;  // if TRUE, the instance afterwards gets moved into the copy code (online change)
	Config : ArduinoLightConfig;
END_VAR
IF Config.IsEnabled THEN
	_config := Config;
	
	SUPER^._lightConfig.Name := Config.Name;
	SUPER^._lightConfig.DeviceID := Config.DeviceID;
	SUPER^._lightConfig.IsEnabled := Config.IsEnabled;
	SUPER^._lightConfig.LogLevel := Config.LogLevel;
	
	SUPER^.Name := Config.Name;
	SUPER^.DeviceID := Config.DeviceID;	
	THIS^.Family := DeviceFamily.Light;
		
	_Logger.Information(_message.Reset().Append('Init ').
							Append('{').Append(TO_STRING(THIS^.Family)).Append('} - ').
							Append('{').Append(TO_STRING(Config.Name)).Append('}').ToString());																													
END_IF
END_METHOD

{attribute 'TcRpcEnable' := '1'}
METHOD GetIntensity
VAR_INPUT
	Execute : BOOL;
	LightId : STRING;
END_VAR
VAR
	cmd : STRING := '*amps ';
END_VAR
IF Execute THEN	
	_deliverMessages := EFeedbackMsgArduinoLight.IntensityMsg;
	_lightId := LightId;
	_serialCom.Send(CONCAT(cmd, TO_STRING(_lightId)));
	
	_getIntensityCmd := FALSE;
END_IF
END_METHOD

METHOD GetLightSources
VAR_INPUT
	Execute: BOOL;
END_VAR
VAR
	cmd : STRING := '*list';
END_VAR
IF Execute THEN
	_logger.Information(_message.Reset().Append(_config.Name).Append(' - GetLightSources').ToString());
	_deliverMessages := EFeedbackMsgArduinoLight.LightSourcesMsg;
	_serialCom.Send(cmd);	
	
	_getLightSourcesCmd := FALSE;
END_IF
END_METHOD

{attribute 'TcRpcEnable' := '1'}
METHOD GetPower
VAR_INPUT
	Execute : BOOL;
	LightId : STRING;
END_VAR
VAR
	cmd : STRING := '*power ';
END_VAR
IF Execute THEN	
	_deliverMessages := EFeedbackMsgArduinoLight.PowerMsg;
	_lightId := LightId;
	_serialCom.Send(CONCAT(cmd, TO_STRING(_lightId)));
	
	 _getPowerCmd := FALSE;
END_IF
END_METHOD

{attribute 'TcRpcEnable' := '1'}
METHOD GetSwitchOn
VAR_INPUT
	Execute : BOOL;
	LightId : STRING;
END_VAR
VAR
	cmd : STRING := '*swit ';
END_VAR
IF Execute THEN	
	_deliverMessages := EFeedbackMsgArduinoLight.SwitchOnMsg;
	_lightId := LightId;
	_serialCom.Send(CONCAT(cmd, TO_STRING(_lightId)));
				
	_getSwitchOnCmd := FALSE;	
END_IF
END_METHOD

METHOD GetTemperature
VAR_INPUT
	LightId : STRING;
END_VAR
VAR
	cmd : STRING := '*temp ';
END_VAR
_deliverMessages := EFeedbackMsgArduinoLight.TemperatureMsg;
_lightId := LightId;
_serialCom.Send(CONCAT(cmd, _lightId));
END_METHOD

METHOD GetTimeLightSource
VAR_INPUT
	Execute: BOOL;
	LightId : STRING;
END_VAR
VAR
	cmd : STRING := '*time ';
END_VAR
IF Execute THEN
	_lightId := LightId;
	_logger.Information(_message.Reset().Append(_config.Name).Append(' - GetTimeLightSource - ').Append(TO_STRING(_lightId)).ToString());
	_deliverMessages := EFeedbackMsgArduinoLight.TimeLightSourceMsg;
	_serialCom.Send(CONCAT(cmd, _lightId));	
	
	_getTimeLightSourceCmd := FALSE;
END_IF
END_METHOD

PROPERTY InitConfigSerialCom : BOOL
GET
InitConfigSerialCom := _initConfigSerialCom;
END_GET
SET
_initConfigSerialCom := InitConfigSerialCom;
END_SET
END_PROPERTY

METHOD InitDevice
VAR_INPUT
END_VAR
VAR
	numElements : INT := 0;
    commaPos : INT;
    tempStr : STRING; 
	Separator : STRING := ',';
END_VAR
IF NOT _initDevice THEN	
	IF _initPulseGenerator.Q THEN
		_initPulseGenerator(IN := FALSE, PT := T#10MS);
			
		CASE _itemInitScheduler OF					
			0:	_logger.Information(_message.Reset().Append(_config.Name).Append(' - Init device').ToString());
				//_getLightSourcesCmd := TRUE;
				_itemInitScheduler := 50;
			
			1:	IF LightSourcesMsg <> '' THEN				
					tempStr := LightSourcesMsg;
					WHILE (LEN(tempStr) > 0) DO
						commaPos := FIND(tempStr, Separator);
						IF commaPos > 0 THEN
							_lightSources[numElements] := LEFT(tempStr, commaPos - 1);						
							tempStr := RIGHT(tempStr, LEN(tempStr) - commaPos);
						ELSE
							_lightSources[numElements] := tempStr;
							tempStr := ''; 
						END_IF
						_logger.Information(_message.Reset().Append(_config.Name).Append(' - ').Append(TO_STRING(numElements)).Append(': ').Append(_lightSources[numElements]).ToString());
						numElements := numElements + 1;						
					END_WHILE
														
					IF (numElements - 1) <> 0 THEN
						_numberOfElements := numElements;
						//_itemInitScheduler := 10; GVA
						_itemInitScheduler := 50;
					ELSE
						_itemInitScheduler := 40;	
					END_IF				
					
					_deliverMessages := -1;
				END_IF
			
			10: IF (_indexNumberOfElements >= 0) AND (_indexNumberOfElements < _numberOfElements) THEN
					tempStr := CONCAT(_lightSources[_indexNumberOfElements], ' 0');
					_serialCom.Send(CONCAT('*power ', tempStr));				
					_logger.Information(_message.Reset().Append(_config.Name).Append(' - ').Append(_lightSources[_indexNumberOfElements]).Append(' - Power: 0').ToString());	
					_indexNumberOfElements := _indexNumberOfElements + 1;
					
				ELSE
					_indexNumberOfElements := 0;
					_itemInitScheduler := 11;					
				END_IF	
			
			11: IF (_indexNumberOfElements >= 0) AND (_indexNumberOfElements < _numberOfElements) THEN
					tempStr := CONCAT(_lightSources[_indexNumberOfElements], ' 1');
					_serialCom.Send(CONCAT('*swit ', tempStr));
					_logger.Information(_message.Reset().Append(_config.Name).Append(' - ').Append(_lightSources[_indexNumberOfElements]).Append(' - Switch ON').ToString());
					_indexNumberOfElements := _indexNumberOfElements + 1;					
				ELSE
					_indexNumberOfElements := 0;
					_itemInitScheduler := 50;
				END_IF	

			41: _logger.Error(_message.Reset().Append(_config.Name).Append(' - numElements is empty: ').ToString());
				_itemInitScheduler := 50;	
		
			50: _initDevice := TRUE;
				_itemInitScheduler := 0;	
				_logger.Information(_message.Reset().Append(_config.Name).Append(' - Init device done').ToString());	
		END_CASE
	ELSE
		_initPulseGenerator(IN := TRUE, PT := T#100MS);		
	END_IF	
END_IF
END_METHOD

METHOD MessageScheduler
VAR_INPUT
END_VAR
IF _pulseGenerator.Q THEN
	_pulseGenerator(IN := FALSE, PT := T#10MS);
		
	CASE _itemScheduler OF					
		0:	IF _lightID <> '' THEN
				//GetTemperature(_lightID);
			END_IF
				
			_itemScheduler := 0;		
	END_CASE
ELSE
	_pulseGenerator(IN := TRUE, PT := T#100MS);		
END_IF


IF _pulseIsAliveGenerator.Q THEN
	_pulseIsAliveGenerator(IN := FALSE, PT := T#10MS);
		
	IsAlive();	
ELSE
	_pulseIsAliveGenerator(IN := TRUE, PT := T#1000MS);		
END_IF
END_METHOD

{attribute 'TcRpcEnable' := '1'}
METHOD RaisePropertiesChanged
VAR_INPUT
	Execute : BOOL;
	LightId : STRING;
END_VAR
VAR
	numElements : INT := 0;
    commaPos : INT;
    tempStr : STRING; 
	Separator : STRING := ',';
END_VAR
IF Execute THEN
	_raisePropertiesCmd := TRUE;
	_lightId := LightId;
	
	IF _pulseGenerator.Q THEN
		_pulseGenerator(IN := FALSE, PT := T#10MS);	

		CASE _itemRaisedProperties OF
			0:  SwitchOnMsg := ' ';
				PowerMsg := ' ';		
				IntensityMsg := ' ';
				LightSourcesMsg := ' ';		
				TimeLightSourceMsg := ' ';		
				_itemRaisedProperties := 1;					

			1:  IF _lightId <> '' THEN
					_itemRaisedProperties := 10;	
				ELSE
					_itemRaisedProperties := 40;	
				END_IF
				
			10: _getSwitchOnCmd := TRUE;													
				_itemRaisedProperties := 11;
				
			11: IF SwitchOnMsg <> ' ' THEN
					_itemRaisedProperties := 12;
				END_IF	
				
			12: _getPowerCmd := TRUE;													
				_itemRaisedProperties := 13;
				
			13: IF PowerMsg <> ' ' THEN
					_itemRaisedProperties := 14;
				END_IF
				
			14: _getIntensityCmd := TRUE;													
				_itemRaisedProperties := 15;
				
			15: IF IntensityMsg <> ' ' THEN
					_itemRaisedProperties := 16;
				END_IF
			
			16: _getTimeLightSourceCmd := TRUE;													
				_itemRaisedProperties := 17;
				
			17: IF TimeLightSourceMsg <> ' ' THEN
					_itemRaisedProperties := 50;
				END_IF
			
			40: _logger.Error(_message.Reset().Append(_config.Name).Append(' - RaisePropertiesChanged - LightId is empty').ToString());
				_itemRaisedProperties := 50;
			
			50:  _logger.Information(_message.Reset().Append(_config.Name).Append(' - RaisePropertiesChanged').ToString());
				_raisePropertiesCmd := FALSE;				
				_itemRaisedProperties := 0;
			
		END_CASE
	ELSE
		_pulseGenerator(IN := TRUE, PT := T#50MS);	
	END_IF
END_IF
END_METHOD

{attribute 'TcRpcEnable' := '1'}
METHOD SetIntensity
VAR_INPUT
	Execute : BOOL;
	LightId : STRING;
	Intensity : LREAL;
END_VAR
VAR
	cmd : STRING := '*amps ';
	tmpConcatLightIdIntensity : STRING;
END_VAR
IF Execute THEN	
	_setIntensityCmd := TRUE;
	_lightId := LightId;
	_setIntensity := Intensity; 
	
	IF _execPulseGenerator.Q THEN
		_execPulseGenerator(IN := FALSE, PT := T#10MS);
			
		CASE _itemExecScheduler OF
			0:  IF _lightId <> '' THEN
					_itemExecScheduler := 10;	
				ELSE
					_itemExecScheduler := 40;	
				END_IF
				
				_deliverMessages := -1;

			10: _lightId := LightId;
				tmpConcatLightIdIntensity := CONCAT(CONCAT(_lightId, ' '), TO_STRING(Intensity));

				_logger.Information(_message.Reset().Append(_config.Name).Append(' - ').Append(_lightId).Append(' - SetIntensity : ').Append(TO_STRING(_lightId)).Append(' - ').Append(TO_STRING(Intensity)).ToString());
				_serialCom.Send(CONCAT(cmd, TO_STRING(tmpConcatLightIdIntensity)));
				_itemExecScheduler := 11;
			
			11:  _getIntensityCmd := TRUE;
				_itemExecScheduler := 50;
			
			40: _logger.Error(_message.Reset().Append(_config.Name).Append(' - SetIntensity - LightId is empty').ToString());
				_itemExecScheduler := 50;
		
			50:  _setIntensityCmd := FALSE;	
				_itemExecScheduler := 0;		
								
		END_CASE
	ELSE
		_execPulseGenerator(IN := TRUE, PT := T#100MS);	
	END_IF
END_IF
END_METHOD

{attribute 'TcRpcEnable' := '1'}
METHOD SetPower
VAR_INPUT
	Execute : BOOL;
	LightId : STRING;
	Power : LREAL;
END_VAR
VAR
	cmd : STRING := '*power ';
	tmpConcatLightIdPower : STRING;
END_VAR
IF Execute THEN	
	_setPowerCmd := TRUE;	
	_lightId := LightId;
	_setPower := Power;	
	
	IF _execPulseGenerator.Q THEN
		_execPulseGenerator(IN := FALSE, PT := T#10MS);
			
		CASE _itemExecScheduler OF
			0:  IF _lightId <> '' THEN
					_itemExecScheduler := 10;	
				ELSE
					_itemExecScheduler := 40;	
				END_IF
				
				_deliverMessages := -1;

			10: _lightId := LightId;
				tmpConcatLightIdPower := CONCAT(CONCAT(_lightId, ' '), TO_STRING(Power));

				_logger.Information(_message.Reset().Append(_config.Name).Append(' - ').Append(_lightId).Append(' - SetPower : ').Append(TO_STRING(Power)).ToString());
				_serialCom.Send(CONCAT(cmd, TO_STRING(tmpConcatLightIdPower)));
				_itemExecScheduler := 11;
			
			11:  _getPowerCmd := TRUE;
				_itemExecScheduler := 50;
			
			40: _logger.Error(_message.Reset().Append(_config.Name).Append(' - SetPower - LightId is empty').ToString());
				_itemExecScheduler := 50;
	
			50:  _setPowerCmd := FALSE;	
				_itemExecScheduler := 0;		
								
		END_CASE
	ELSE
		_execPulseGenerator(IN := TRUE, PT := T#100MS);	
	END_IF
END_IF
END_METHOD

{attribute 'TcRpcEnable' := '1'}
METHOD SetSwitchOn
VAR_INPUT
	Execute : BOOL;	
	LightId : STRING;
	SwitchOn : BOOL;
END_VAR
VAR
	cmd : STRING := '*swit ';
	tmpConcatLightIdSwitchOn : STRING;
	tmp : STRING;
	switchOnValue : STRING;
END_VAR
IF Execute THEN	
	_setSwitchOnCmd := TRUE;	
	_switchOn := SwitchOn; 
	_lightId := LightId;
	
	IF _execPulseGenerator.Q THEN
		_execPulseGenerator(IN := FALSE, PT := T#10MS);
			
		CASE _itemExecScheduler OF
			0:  IF _lightId <> '' THEN
					_itemExecScheduler := 10;	
				ELSE
					_itemExecScheduler := 40;	
				END_IF
				
				_deliverMessages := -1;

			10:	_lightId := LightId;				
			
				IF _switchOn THEN
					switchOnValue := '1';
				ELSE
					switchOnValue := '0';
				END_IF
				tmpConcatLightIdSwitchOn := CONCAT(CONCAT(_lightId, ' '), TO_STRING(switchOnValue));
				
				_logger.Information(_message.Reset().Append(_config.Name).Append(' - ').Append(_lightId).Append(' - SwitchOn : ').Append(TO_STRING(switchOnValue)).ToString());
				tmp := CONCAT(cmd, TO_STRING(tmpConcatLightIdSwitchOn));
				_serialCom.Send(tmp);
				_itemExecScheduler := 11;
			
			11:  _getSwitchOnCmd := TRUE;
				_itemExecScheduler := 50;
				
			40: _logger.Error(_message.Reset().Append(_config.Name).Append(' - SwitchOn - LightId is empty').ToString());
				_itemExecScheduler := 50;
				
			50:  _setSwitchOnCmd := FALSE;	
				_switchOn := FALSE;
				_itemExecScheduler := 0;		
								
		END_CASE
	ELSE
		_execPulseGenerator(IN := TRUE, PT := T#200MS);	
	END_IF
END_IF
END_METHOD

END_FUNCTION_BLOCK

// ---- Service/PMs/PhotoLum/Communication/RS232/PhotoLumBkgrdSerialCom.TcPOU
PROGRAM PhotoLumBkgrdSerialCom
VAR_INPUT
	Config : PhotoLumConfig;
END_VAR
VAR
END_VAR

// AxisConfigs
IF Config.AxesConfigs.Ps10OwisAxisConfig.IsEnabled THEN
	BkgrdSerialOwisPs10();	
END_IF

// LightConfigs
IF Config.LightConfigs.ArduinoLightConfig.IsEnabled THEN
	BkgrdSerialLight();
ELSIF Config.LightConfigs.EvosensLightConfig.IsEnabled THEN
	BkgrdSerialLight();
END_IF

END_PROGRAM

// ---- PMShared/Hardware/Devices/Axes/Configs/Owis/SerialCommunication/BkgrdSerialOwisPs10.TcPOU
PROGRAM BkgrdSerialOwisPs10
VAR
	(* background communication with the EL6002 terminal *)
	serialLineCtrl		: SerialLineControl;
	serialLineCtrlError	: BOOL;
	serialLineCtrlErrorID : ComError_t;
	(* 	I/O variables for a EL6002 terminal*)
	stInFilterWheel  AT %I*	: EL6inData22B;	
	stOutFilterWheel AT %Q*	: EL6outData22B;
END_VAR

(*
The SerialLineControl function block is supposed to be called in every PLC cycle.
It communicates with the serial line hardware device and transmits or receives data.
The SerialLineControl can be called in the standard task (e.g.for PcCOM port usage) 
or in a separate fast task (e.g.for terminal usage) as well.
A fast separate task will be necessary at high baud rates or with KL6001 terminals 
which have a small process image (3 or 5 data bytes only)
*)

(* background communication with the EL6002 terminal *)
serialLineCtrl(
	Mode:= SERIALLINEMODE_EL6_22B, 
	pComIn:= ADR(stInFilterWheel), 
	pComOut:= ADR(stOutFilterWheel), 
	SizeComIn:= SIZEOF(stInFilterWheel), 
	TxBuffer:= HardwareGlobalVariables.TxBufferFilterWheel, 
	RxBuffer:= HardwareGlobalVariables.RxBufferFilterWheel
);

IF serialLineCtrl.Error THEN
	serialLineCtrlError := TRUE;
	serialLineCtrlErrorID := serialLineCtrl.ErrorID;
END_IF

END_PROGRAM

// ---- PMShared/Hardware/Devices/Lights/Configs/SerialCommunication/BkgrdSerialLight.TcPOU
PROGRAM BkgrdSerialLight
VAR
	(* background communication with the EL6002 terminal *)
	serialLineCtrl		: SerialLineControl;
	serialLineCtrlError	: BOOL;
	serialLineCtrlErrorID : ComError_t;
	(* 	I/O variables for a EL6002 terminal*)
	stInLight  AT %I* : EL6inData22B;	
	stOutLight AT %Q* : EL6outData22B;
END_VAR

(*
The SerialLineControl function block is supposed to be called in every PLC cycle.
It communicates with the serial line hardware device and transmits or receives data.
The SerialLineControl can be called in the standard task (e.g.for PcCOM port usage) 
or in a separate fast task (e.g.for terminal usage) as well.
A fast separate task will be necessary at high baud rates or with KL6001 terminals 
which have a small process image (3 or 5 data bytes only)
*)

(* background communication with the EL6002 terminal *)
serialLineCtrl(
	Mode:= SERIALLINEMODE_EL6_22B, 
	pComIn:= ADR(stInLight), 
	pComOut:= ADR(stOutLight), 
	SizeComIn:= SIZEOF(stInLight), 
	TxBuffer:= HardwareGlobalVariables.TxBufferLight, 
	RxBuffer:= HardwareGlobalVariables.RxBufferLight
);

IF serialLineCtrl.Error THEN
	serialLineCtrlError := TRUE;
	serialLineCtrlErrorID := serialLineCtrl.ErrorID;
END_IF

END_PROGRAM

// ---- PMShared/Hardware/Common/Tools/PWM/PwmGenerator.TcPOU
FUNCTION_BLOCK PUBLIC PwmGenerator
VAR_INPUT
	
END_VAR
VAR_OUTPUT
	
END_VAR
VAR_IN_OUT
   StParams : ST_CTRL_PWM_OUT_PARAMS;
END_VAR
VAR
	{region 'FB_CTRL_PWM_OUT'}		
	_pwm : FB_CTRL_PWM_OUT;
	
	fPwmInput : LREAL := 1;
   	eMode     : E_CTRL_MODE;
	bPwmOutBitPos : BOOL;       
	bPwmOutBitNeg : BOOL;       
	eState		 : E_CTRL_STATE;
	_pwmError    : BOOL;
	_pwmErrorId  : E_CTRL_ERRORCODES;
	{endregion}
		 
END_VAR



_pwm(
	fPwmInput:= fPwmInput ,
	eMode:= E_CTRL_MODE.eCTRL_MODE_MANUAL,
	stParams:= StParams,
	bPwmOutBitPos=> bPwmOutBitPos,
	bPwmOutBitNeg=> bPwmOutBitNeg,
	eState=> eState,
	eErrorId=> _pwmErrorId,
	bError=> _pwmError);

END_FUNCTION_BLOCK

// ---- Shared/Tools/Trigger/Trigger.TcPOU
FUNCTION_BLOCK PUBLIC Trigger
VAR_INPUT
END_VAR
VAR_OUTPUT
END_VAR
VAR
	{attribute 'OPC.UA.DA' := '0'}
	_logger : Logger;
	{attribute 'OPC.UA.DA' := '0'}
	_message : StringBuilder;
	
	{attribute 'OPC.UA.DA' := '0'}
	_execStartTrigger : BOOL;

	{attribute 'OPC.UA.DA' := '0'}
	_stateCmd : INT;
	{attribute 'OPC.UA.DA' := '0'}
	_setPeriod_ms : LREAL;
	
	{attribute 'OPC.UA.DA' := '0'}
	timerDelayOn : TON;
	{attribute 'OPC.UA.DA' := '0'}
	timerDelayOff: TON;	
	{attribute 'OPC.UA.DA' := '0'}
	pulseFlag : BOOL;
	{attribute 'OPC.UA.DA' := '0'}	
	trigOff : BOOL;	
	{attribute 'OPC.UA.DA' := '0'}
	OutputTrigger	AT %Q* : BOOL;	
END_VAR

TriggerOutEmitSignal(_execStartTrigger, _setPeriod_ms);

{attribute 'TcRpcEnable' := '1'}
METHOD PROTECTED TriggerOutEmitSignal
VAR_INPUT
	Execute : BOOL;
	PulseDuration_ms : LREAL;	
END_VAR
VAR
	demiPulseDuration_ms : TIME;
END_VAR
(*
// La FastTask a un cycle de 50µs. Il faut 4 instructions pour obtenir un pulse.
// On aura donc un pulse minimum de 200 µs (4 * 50 µs) 
*)

IF Execute THEN
	_execStartTrigger := TRUE;
	_setPeriod_ms := PulseDuration_ms;
	
	demiPulseDuration_ms := LREAL_TO_TIME(_setPeriod_ms * 1E+6) / 2;
	
	_logger.Information(_message.Reset().Append('TriggerOutEmitSignal').ToString());
	
	CASE _stateCmd OF
		0:  timerDelayOn(IN := _execStartTrigger AND NOT trigOff, PT := demiPulseDuration_ms);
			OutputTrigger := timerDelayOn.Q;
			
			timerDelayOff(IN := OutputTrigger, PT := demiPulseDuration_ms);
			trigOff := timerDelayOff.Q;
				
			//_execStartTrigger := FALSE;
	END_CASE
END_IF
END_METHOD

END_FUNCTION_BLOCK

// ---- PMShared/Hardware/Devices/Axes/IoAxis/Stage/IoStageAxis.TcPOU
FUNCTION_BLOCK IoStageAxis EXTENDS AxesBase
VAR_INPUT
END_VAR
VAR_OUTPUT
END_VAR
VAR
	{attribute 'OPC.UA.DA' := '0'}
	_config : IoStageAxisConfig;
	{attribute 'OPC.UA.DA' := '0'}
	IoStageStruct : IoStageStruct;
	
	{attribute 'OPC.UA.DA' := '0'}
	_deliverMessages : INT;
	
	PositionMsg : STRING(255);
	
	{region 'Commands'}	
		 
	{attribute 'OPC.UA.DA' := '0'}
	_moveAbsPosition	 : BOOL;
	{attribute 'OPC.UA.DA' := '0'}			  		   
	_raiseProperties : BOOL;	 
			
	{endregion}
		 
	{attribute 'OPC.UA.DA' := '0'}
	_initDevice : BOOL;	
		
	{attribute 'OPC.UA.DA' := '0'}
	_pos : INT; //EPosition;
	{attribute 'OPC.UA.DA' := '0'}
	_itemScheduler : INT;
	{attribute 'OPC.UA.DA' := '0'}
	_itemRaisedProperties : INT;
	{attribute 'OPC.UA.DA' := '0'}
	_pulseGenerator : TON;
END_VAR


// Init device
InitDevice(); 

// Deliver messages
CASE _deliverMessages OF	
	EFeedbackMsgStage.PositionMsg :
		PositionMsg := INT_TO_STRING(GetPosition());			
END_CASE
	
_deliverMessages := 0;

// Commands
MoveAbsPosition(_moveAbsPosition, _pos); 
RaisePropertiesChanged(_raiseProperties);

IF (NOT _moveAbsPosition AND NOT _raiseProperties) THEN
	MessageScheduler();
END_IF

METHOD FB_init : BOOL
VAR_INPUT
	bInitRetains : BOOL; // if TRUE, the retain variables are initialized (warm start / cold start)
	bInCopyCode : BOOL;  // if TRUE, the instance afterwards gets moved into the copy code (online change)
	Config : IoStageAxisConfig;
END_VAR
IF Config.IsEnabled THEN
	_config := Config;
	
	SUPER^._axisConfig.Name := Config.Name;
	SUPER^._axisConfig.DeviceID := Config.DeviceID;
	SUPER^._axisConfig.IsEnabled := Config.IsEnabled;
	SUPER^._axisConfig.LogLevel := Config.LogLevel;
	
	SUPER^.Name := Config.Name;
	SUPER^.DeviceID := Config.DeviceID;	
	THIS^.Family := DeviceFamily.Axes;
	
	_Logger.Information(_message.Reset().Append('Init ').
							Append('{').Append(TO_STRING(THIS^.Family)).Append('} - ').
							Append('{').Append(TO_STRING(Config.Name)).Append('}').ToString());																													
END_IF
END_METHOD

METHOD GetPosition : INT
VAR_INPUT
END_VAR
_deliverMessages := EFeedbackMsgStage.PositionMsg;

IF IsStageInProcessPosition(IoStageStruct.InputProcessPosition) THEN
	GetPosition := EStagePosition.Process;
ELSIF IsStageInProcessPosition(IoStageStruct.InputLoadingPosition) THEN
	GetPosition := EStagePosition.Loading;
ELSE
	GetPosition := EStagePosition.Unknown;		
END_IF
END_METHOD

METHOD InitDevice : BOOL
VAR_INPUT
END_VAR
IF NOT _initDevice THEN	
	_logger.Information(_message.Reset().
								Append(_config.Name).
								Append(' - Init device').ToString());
							
	THIS^.Status := TExecutionState.Ready;
	
	GetPosition();
	
	_initDevice := TRUE;	
END_IF
END_METHOD

METHOD IsStageInLoadingPosition : BOOL
VAR_INPUT
	Position : INT;
END_VAR
VAR
	val : INT; 
END_VAR
val := ABS(Position - Const.FLEXO_AI_PISTON_LEFT_SENSING_RANGE_MAX);

IF val < Const.FLEXO_AI_PISTON_LEFT_SENSING_RANGE_MIN THEN
	IsStageInLoadingPosition := TRUE;
ELSE
	IsStageInLoadingPosition := FALSE;
END_IF
END_METHOD

METHOD IsStageInProcessPosition : BOOL
VAR_INPUT
	Position : INT;
END_VAR
VAR
	val : INT; 
END_VAR
val := ABS(Position - Const.FLEXO_AI_PISTON_LEFT_SENSING_RANGE_MAX);

IF val < Const.FLEXO_AI_PISTON_LEFT_SENSING_RANGE_MIN THEN
	IsStageInProcessPosition := TRUE;
ELSE
	IsStageInProcessPosition := FALSE;
END_IF
END_METHOD

METHOD MessageScheduler
VAR_INPUT
END_VAR
IF _pulseGenerator.Q THEN
	_pulseGenerator(IN := FALSE, PT := T#10MS);
		
	CASE _itemScheduler OF	
		0:	GetPosition();
			_itemScheduler := 0;										
	END_CASE
ELSE
	_pulseGenerator(IN := TRUE, PT := T#100MS);	
END_IF
END_METHOD

{attribute 'TcRpcEnable' := '1'}
METHOD PROTECTED MoveAbsPosition 
VAR_INPUT
	Execute : BOOL;
	Position : LREAL;
END_VAR
VAR	
END_VAR
IF Execute THEN
	_logger.Information(_message.Reset().Append(_config.Name).Append(' - Move absolute position : ').Append(TO_STRING(Position)).ToString());
	
	_moveAbsPosition := FALSE;	
	
	IF Position = EStagePosition.Loading THEN
		IoStageStruct.OutputLoadingPosition := FALSE;
		IoStageStruct.OutputProcessPosition := TRUE;		
	ELSIF Position = EStagePosition.Process THEN
		IoStageStruct.OutputLoadingPosition := TRUE;
		IoStageStruct.OutputProcessPosition := FALSE;
	ELSE
		_logger.Error(_message.Reset().Append(_config.Name).Append(' - unknown position : ').Append(TO_STRING(Position)).ToString());								
	END_IF
			
	_itemScheduler := 0;
END_IF
END_METHOD

{attribute 'TcRpcEnable' := '1'}
METHOD RaisePropertiesChanged
VAR_INPUT
	Execute : BOOL;
END_VAR
IF Execute THEN		
	_raiseProperties := TRUE;	
	
	IF _pulseGenerator.Q THEN
		_pulseGenerator(IN := FALSE, PT := T#10MS);
		
		CASE _itemRaisedProperties OF		
			0: PositionMsg := ' ';
				_itemRaisedProperties := 1;
			
			1: GetPosition();		   
				_itemRaisedProperties := 10;
				
			10: 
				_logger.Information(_message.Reset().
								    Append(_config.Name).
								    Append(' - RaisePropertiesChanged').ToString());
				_raiseProperties := FALSE;
				_itemRaisedProperties := 0;
		
		END_CASE
	
	ELSE
		_pulseGenerator(IN := TRUE, PT := T#50MS);	
	END_IF
		
END_IF
END_METHOD

METHOD ReadStagePosition
VAR_INPUT
END_VAR
END_METHOD

END_FUNCTION_BLOCK
